DATA_BLOCK "dbMasterData"   // DB35
{ S7_Optimized_Access := 'FALSE' }
VERSION : 0.1
// stored: AutoNumber false, DBAccessibleFromOPCUA true, IsOnlyStoredInLoadMemory false, IsWriteProtectedInAS false
   VAR
      data5_Wielkość_przeływu_Adres_0 { S7_SetPoint := 'True'} : "typeDataMPP04_Int";   // wielkość przepływu / Wartość aktualnego przepływu
      data5_Licznik_objętość_VF_Adres_2 : "typeDataMPP04_Int";   // licznik objętości VF / Stan licznika objętości dla przepływu w przód VF
      data5_Licznik_objętość_VR_Adres_4 { S7_SetPoint := 'True'} : "typeDataMPP04_Int";   // licznik objętości VR / Stan licznika objętości dla przepływu w tył VR
      data5_Licznik_różnicowy_VD_Adres_6 { S7_SetPoint := 'True'} : "typeDataMPP04_Int";   // licznik różnicy / Stan bieżącego różnicowego licznika objętości VD
      data5_Stan_licz_bjętości_GF_Adres_8 { S7_SetPoint := 'True'} : "typeDataMPP04_Int";   // licznik objetosci GF / Stan głównego licznika objętości dla przepływu w przód GF
      data5_Stan_licz_bjętości_GR_Adres_10 { S7_SetPoint := 'True'} : "typeDataMPP04_Int";   // licznik objetości GR / Sta ngłownego licznika objętości dla przepływu w tył GR
      data5_Stan_licz_rózicowego_obj_GD_Adres_12 { S7_SetPoint := 'True'} : "typeDataMPP04_Int";   // licznik róznicowy / Stan głownego licznika różnicowego GD
      data5_Stan_urządzenia_1000 { S7_SetPoint := 'True'} : "typeDataInverter_Word";   // stan urządzenia / 8-przekrodzony zakres pracy przetwornika, 20-otwarty obwód cewki, 21zwarcie w obwodzie cewki, 26-brak cieczy w czujniku
      data6_Wielkość_przeływu_Adres_0 { S7_SetPoint := 'True'} : "typeDataMPP04_Int";   // wielkość przepływu / Wartość aktualnego przepływu
      data6_Licznik_objętość_VF_Adres_2 { S7_SetPoint := 'True'} : "typeDataMPP04_Int";   // licznik objętości VF / Stan licznika objętości dla przepływu w przód VF
      data6_Licznik_objętość_VR_Adres_4 { S7_SetPoint := 'True'} : "typeDataMPP04_Int";   // licznik objętości VR / Stan licznika objętości dla przepływu w tył VR
      data6_Licznik_różnicowy_VD_Adres_6 { S7_SetPoint := 'True'} : "typeDataMPP04_Int";   // licznik różnicy / Stan bieżącego różnicowego licznika objętości VD
      data6_Stan_licz_bjętości_GF_Adres_8 { S7_SetPoint := 'True'} : "typeDataMPP04_Int";   // licznik objetosci GF / Stan głównego licznika objętości dla przepływu w przód GF
      data6_Stan_licz_bjętości_GR_Adres_10 { S7_SetPoint := 'True'} : "typeDataMPP04_Int";   // licznik objetości GR / Sta ngłownego licznika objętości dla przepływu w tył GR
      data6_Stan_licz_rózicowego_obj_GD_Adres_12 { S7_SetPoint := 'True'} : "typeDataMPP04_Int";   // licznik róznicowy / Stan głownego licznika różnicowego GD
      data6_Stan_urządzenia_1000 { S7_SetPoint := 'True'} : "typeDataInverter_Word";   // stan urządzenia / 8-przekrodzony zakres pracy przetwornika, 20-otwarty obwód cewki, 21zwarcie w obwodzie cewki, 26-brak cieczy w czujniku
      data26_Inver_Control_word_416000_Fal { S7_SetPoint := 'True'} : "typeDataInverter_Word";   // Sowo komtrolneCTW falownika [Uint16, index 0]
      data26_Inver_setpoint_ref_416020_Fal { S7_SetPoint := 'True'} : "typeDataInverter_Word";   // Słowo wartość zadana Hz [Int16, index -1]
      data26_Inver_Status_word_416030_Fal { S7_SetPoint := 'True'} : "typeDataInverter_Word";   // Słowo statusu STW falownika [Uint16, index 0]
      data26_Inver_Frequency_416130_Fal { S7_SetPoint := 'True'} : "typeDataInverter_Word";   // Słowo częstotliwość na wyjściu [Uint16, index -1]
      data26_Inver_MotorCurrent_416140_Fal { S7_SetPoint := 'True'} : "typeDataInverter_Word";   // Słowo częstotliwość na wyjściu [Uint16, index -2]
      data26_Inver_DC_Voltage_416300_Fal { S7_SetPoint := 'True'} : "typeDataInverter_Word";   // Słowo napięcia DC na szynie [Uint16, index 0]
      data26_Inver_Temp_416340_Fal { S7_SetPoint := 'True'} : "typeDataInverter_Word";   // Słowo temperatura invertera [Uint8, index 0]
      data26_Inver_NomCurrent_416360_Fal { S7_SetPoint := 'True'} : "typeDataInverter_Word";   // Słowo nominalna wartośc prądu falonika[Uint16, index -2]
      data26_Inver_MaxCurrent_416370_Fal { S7_SetPoint := 'True'} : "typeDataInverter_Word";   // Słowo max prąd falownika [Uint16, index -2]
      data26_Inver_InDigit_416600_Fal { S7_SetPoint := 'True'} : "typeDataInverter_Word";   // Słowo mampa wejść 18,19,27,33 [Uint16, index -0]
      data26_Inver_HourWork_415010_Fal { S7_SetPoint := 'True'} : "typeDataInverter_DWord";   // Podwójne słowo czasu pracy falownika [Int32, index -0]
      data26_Inver_OverTemp_415040_Fal { S7_SetPoint := 'True'} : "typeDataInverter_Word";   // Sowo statusu przekroczenie temperatury[Uint16, index 0]
      data26_Inver_OverVolts_415050_Fal { S7_SetPoint := 'True'} : "typeDataInverter_Word";   // Sowo statusu przekroczenie napięcia[Uint16, index 0]
      data_RTU_value_0 { S7_SetPoint := 'True'} : "typeDataMPP04_real";   // Wartość 0.0 pomocnicza wyświetlana podczas błędu pomiaru
   END_VAR
BEGIN
   data_RTU_value_0.data[0] := 0.0;
END_DATA_BLOCK

DATA_BLOCK "dbModbusRTU_Reg"   // DB37
TITLE = Modbus RTU Data
{ S7_Optimized_Access := 'FALSE' }
AUTHOR : RTecmer
VERSION : 0.1
// Dane pomiarowe przekazane z bloku danych master modbus RTU
// stored: AutoNumber true, DBAccessibleFromOPCUA true, IsOnlyStoredInLoadMemory false, IsWriteProtectedInAS false
   VAR
      received_6_Wielkość_przeływu_Adres_0 { S7_SetPoint := 'True'} : "typeDataMPP04_Int";   // wielkość przepływu
      received_6_Licznik_objętość_VF_Adres_2 { S7_SetPoint := 'True'} : "typeDataMPP04_Int";   // licznik objętości VF
      received_6_Licznik_objętość_VR_Adres_4 { S7_SetPoint := 'True'} : "typeDataMPP04_Int";   // licznik objętości VR
      received_6_Licznik_różnicowy_VD_Adres_6 { S7_SetPoint := 'True'} : "typeDataMPP04_Int";   // licznik różnicy
      receive_6_Stan_licz_bjętości_GF_Adres_8 { S7_SetPoint := 'True'} : "typeDataMPP04_Int";   // licznik objetosci GF
      received_6_Stan_licz_bjętości_GR_Adres_10 { S7_SetPoint := 'True'} : "typeDataMPP04_Int";   // licznik objetości GR
      received_6_Stan_licz_rózicowego_obj_GD_Adres_12 { S7_SetPoint := 'True'} : "typeDataMPP04_Int";   // licznik róznicowy
      received_6_Stan_urządzenia_1000 { S7_SetPoint := 'True'} : "typeDataInverter_Word";   // stan urządzenia
      "Przepływomierz nr2" : Struct
         received_6_przeływu_VF_Adres_0 { S7_SetPoint := 'True'} : Real;
         received_6_objętość_VF_Adres_2 { S7_SetPoint := 'True'} : Real;
         "received_6_objętośc RF_Adres_4" { S7_SetPoint := 'True'} : Real;
         received_6_licznik_różnicowy_VD_Adres_7 { S7_SetPoint := 'True'} : Real;
         received_6_licznik_objętości_GF_Adres_8 { S7_SetPoint := 'True'} : Real;
         received_6_Licznik_objętości_GR_Adres_10 { S7_SetPoint := 'True'} : Real;
         received_6_Licznik_różnicowy_GD_Adres_12 { S7_SetPoint := 'True'} : Real;
         received_6_status_przepływomierza_Adres_1000 { S7_SetPoint := 'True'} : Word;
      END_STRUCT;
   END_VAR
BEGIN
END_DATA_BLOCK

DATA_BLOCK "dbTags_master_MPP04_2"   // DB81
{ S7_Optimized_Access := 'FALSE' }
VERSION : 0.1
// stored: AutoNumber true, DBAccessibleFromOPCUA true, IsOnlyStoredInLoadMemory false, IsWriteProtectedInAS false
   VAR
      "step" : USInt := 1;
      edge : Bool := false;
      modbusCommLoad { S7_SetPoint := 'True'} : "typeModbusCommLoad";
      modbusMaster { S7_SetPoint := 'True'} : "typeModbusMaster";
   END_VAR
BEGIN
END_DATA_BLOCK

DATA_BLOCK "dbTags_master_RTU"   // DB90
TITLE = Master
{ S7_Optimized_Access := 'FALSE' }
AUTHOR : rtecmer
VERSION : 0.1
// Instancja dla funkcji Mdbus RTU komunikacja z masterem MT101
// stored: AutoNumber false, DBAccessibleFromOPCUA true, IsOnlyStoredInLoadMemory false, IsWriteProtectedInAS false
   VAR
      "step" : USInt := 1;
      edge : Bool := false;
      modbusCommLoad { S7_SetPoint := 'True'} : "typeModbusCommLoad";
      modbusMaster { S7_SetPoint := 'True'} : "typeModbusSlave";
   END_VAR
BEGIN
   modbusMaster.mbAddr := 5;
END_DATA_BLOCK

ORGANIZATION_BLOCK "Main"   // OB1, LAD, ProgramCycle
TITLE = "Main Program Sweep (Cycle)"
{ S7_Optimized_Access := 'TRUE' }
VERSION : 0.1
// stored: AutoNumber true, IsIECCheckEnabled false, SetENOAutomatically false
   VAR_INPUT
      Initial_Call : Bool;   // Initial call of this OB
      Remanence : Bool;   // =True, if remanent data are available
   END_VAR
   VAR_TEMP   // added for the SCL form of the ladder/FBD networks
      _w1 : Bool;
      _w2 : Bool;
   END_VAR
BEGIN

REGION Network 1: Diagnostyka przerwań
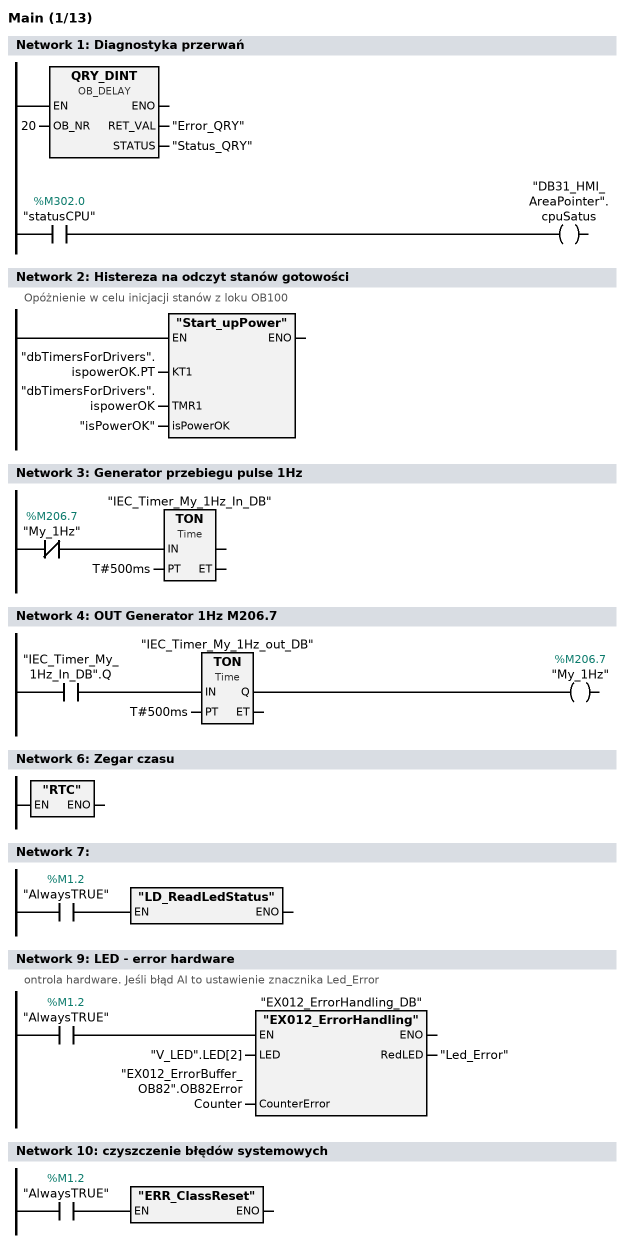
   RUNG wire#powerrail
      { S7_Templates := "obnr_type := OB_DELAY" } QRY_DINT(OB_NR := 20, RET_VAL => "Error_QRY", STATUS => "Status_QRY")
   END_RUNG
   RUNG wire#powerrail
      Contact( "statusCPU" )
      Coil( "DB31_HMI_AreaPointer".cpuSatus )
   END_RUNG
   // the same network as SCL:
   "Error_QRY" := QRY_DINT(OB_NR := 20, STATUS => "Status_QRY");
   "DB31_HMI_AreaPointer".cpuSatus := "statusCPU";
END_REGION

REGION Network 2: Histereza na odczyt stanów gotowości
   // Opóżnienie w celu inicjacji stanów z loku OB100
   RUNG wire#powerrail
      "Start_upPower"(KT1 := "dbTimersForDrivers".ispowerOK.PT, TMR1 := "dbTimersForDrivers".ispowerOK, isPowerOK := "isPowerOK")
   END_RUNG
   // the same network as SCL:
   "Start_upPower"(KT1 := "dbTimersForDrivers".ispowerOK.PT,
                   TMR1 := "dbTimersForDrivers".ispowerOK,
                   isPowerOK := "isPowerOK");
END_REGION

REGION Network 3: Generator przebiegu pulse 1Hz
   RUNG wire#powerrail
      I_Contact( "My_1Hz" )
      { S7_Templates := "time_type := Time" } "IEC_Timer_My_1Hz_In_DB".TON(pt := T#500ms, et =>)
   END_RUNG
   // the same network as SCL:
   "IEC_Timer_My_1Hz_In_DB".TON(IN := NOT "My_1Hz", PT := T#500ms);
END_REGION

REGION Network 4: OUT Generator 1Hz M206.7
   RUNG wire#powerrail
      Contact( "IEC_Timer_My_1Hz_In_DB".Q )
      { S7_Templates := "time_type := Time" } "IEC_Timer_My_1Hz_out_DB".TON(pt := T#500ms, et =>)
      Coil( "My_1Hz" )
   END_RUNG
   // the same network as SCL:
   "IEC_Timer_My_1Hz_out_DB".TON(IN := "IEC_Timer_My_1Hz_In_DB".Q, PT := T#500ms);
   "My_1Hz" := "IEC_Timer_My_1Hz_out_DB".Q;
END_REGION

REGION Network 6: Zegar czasu
   RUNG wire#powerrail
      "RTC"()
   END_RUNG
   // the same network as SCL:
   "RTC"();
END_REGION

REGION Network 7
   RUNG wire#powerrail
      Contact( "AlwaysTRUE" )
      "LD_ReadLedStatus"()
   END_RUNG
   // the same network as SCL:
   IF "AlwaysTRUE" THEN "LD_ReadLedStatus"(); END_IF;
END_REGION

REGION Network 8 (SCL): LED kontrola RUN
   // Przekazanie  stanu LED 1 CPU
   "DB31_HMI_AreaPointer".getPLCMode := "V_LED".LED[1];
END_REGION

REGION Network 9: LED - error hardware
   // ontrola hardware. Jeśli błąd AI to ustawienie znacznika Led_Error
   RUNG wire#powerrail
      Contact( "AlwaysTRUE" )
      "EX012_ErrorHandling_DB"(LED := "V_LED".LED[2], CounterError := "EX012_ErrorBuffer_OB82".OB82ErrorCounter, RedLED => "Led_Error")
   END_RUNG
   // the same network as SCL:
   IF "AlwaysTRUE" THEN
       "EX012_ErrorHandling_DB"(LED := "V_LED".LED[2],   // "EX012_ErrorHandling"
                               CounterError := "EX012_ErrorBuffer_OB82".OB82ErrorCounter,
                               RedLED => "Led_Error");
   END_IF;
END_REGION

REGION Network 10: czyszczenie błędów systemowych
   RUNG wire#powerrail
      Contact( "AlwaysTRUE" )
      "ERR_ClassReset"()
   END_RUNG
   // the same network as SCL:
   IF "AlwaysTRUE" THEN "ERR_ClassReset"(); END_IF;
END_REGION

REGION Network 11: kontrola błedów
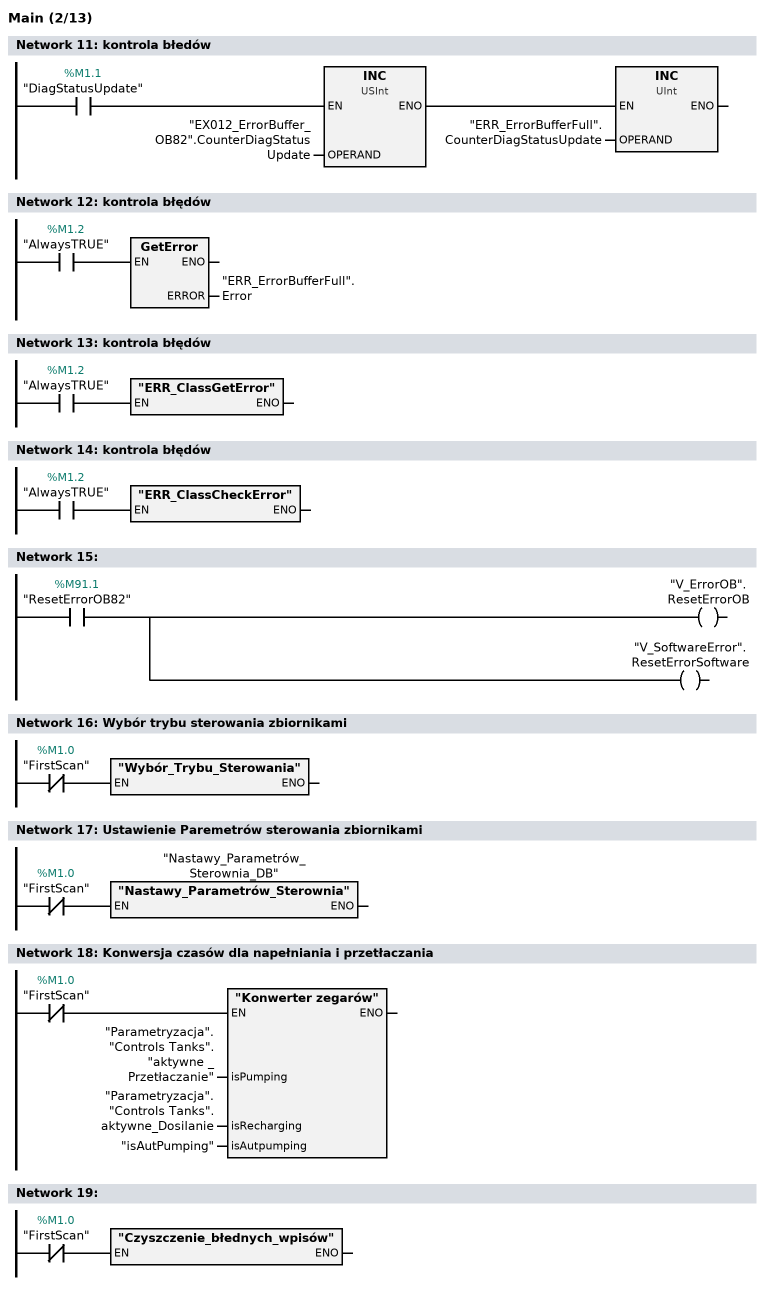
   RUNG wire#powerrail
      Contact( "DiagStatusUpdate" )
      { S7_Templates := "DestType := USInt" } Inc( "EX012_ErrorBuffer_OB82".CounterDiagStatusUpdate )
      { S7_Templates := "DestType := UInt" } Inc( "ERR_ErrorBufferFull".CounterDiagStatusUpdate )
   END_RUNG
   // the same network as SCL:
   IF "DiagStatusUpdate" THEN
       "EX012_ErrorBuffer_OB82".CounterDiagStatusUpdate := "EX012_ErrorBuffer_OB82".CounterDiagStatusUpdate + 1;
       "ERR_ErrorBufferFull".CounterDiagStatusUpdate := "ERR_ErrorBufferFull".CounterDiagStatusUpdate + 1;
   END_IF;
END_REGION

REGION Network 12: kontrola błędów
   // no SCL statement known for GetError: written as a call
   IF "AlwaysTRUE" THEN GetError(error => "ERR_ErrorBufferFull".Error); END_IF;
END_REGION

REGION Network 13: kontrola błędów
   RUNG wire#powerrail
      Contact( "AlwaysTRUE" )
      "ERR_ClassGetError"()
   END_RUNG
   // the same network as SCL:
   IF "AlwaysTRUE" THEN "ERR_ClassGetError"(); END_IF;
END_REGION

REGION Network 14: kontrola błędów
   RUNG wire#powerrail
      Contact( "AlwaysTRUE" )
      "ERR_ClassCheckError"()
   END_RUNG
   // the same network as SCL:
   IF "AlwaysTRUE" THEN "ERR_ClassCheckError"(); END_IF;
END_REGION

REGION Network 15
   RUNG wire#powerrail
      Contact( "ResetErrorOB82" )
      wire#w1
      Coil( "V_ErrorOB".ResetErrorOB )
   END_RUNG
   RUNG wire#w1
      Coil( "V_SoftwareError".ResetErrorSoftware )
   END_RUNG
   // the same network as SCL:
   "V_ErrorOB".ResetErrorOB := "ResetErrorOB82";
   "V_SoftwareError".ResetErrorSoftware := "ResetErrorOB82";
END_REGION

REGION Network 16: Wybór trybu sterowania zbiornikami
   RUNG wire#powerrail
      I_Contact( "FirstScan" )
      "Wybór_Trybu_Sterowania"()
   END_RUNG
   // the same network as SCL:
   IF NOT "FirstScan" THEN "Wybór_Trybu_Sterowania"(); END_IF;
END_REGION

REGION Network 17: Ustawienie Paremetrów sterowania zbiornikami
   RUNG wire#powerrail
      I_Contact( "FirstScan" )
      "Nastawy_Parametrów_Sterownia_DB"()
   END_RUNG
   // the same network as SCL:
   IF NOT "FirstScan" THEN
       "Nastawy_Parametrów_Sterownia_DB"();   // "Nastawy_Parametrów_Sterownia"
   END_IF;
END_REGION

REGION Network 18: Konwersja czasów dla napełniania i przetłaczania
   RUNG wire#powerrail
      I_Contact( "FirstScan" )
      "Konwerter zegarów"(isPumping := "Parametryzacja"."Controls Tanks"."aktywne _Przetłaczanie", isRecharging := "Parametryzacja"."Controls Tanks".aktywne_Dosilanie, isAutpumping := "isAutPumping")
   END_RUNG
   // the same network as SCL:
   IF NOT "FirstScan" THEN
       "Konwerter zegarów"(isPumping := "Parametryzacja"."Controls Tanks"."aktywne _Przetłaczanie",
                           isRecharging := "Parametryzacja"."Controls Tanks".aktywne_Dosilanie,
                           isAutpumping := "isAutPumping");
   END_IF;
END_REGION

REGION Network 19
   RUNG wire#powerrail
      I_Contact( "FirstScan" )
      "Czyszczenie_błednych_wpisów"()
   END_RUNG
   // the same network as SCL:
   IF NOT "FirstScan" THEN "Czyszczenie_błednych_wpisów"(); END_IF;
END_REGION

REGION Network 20: Modbus RTU
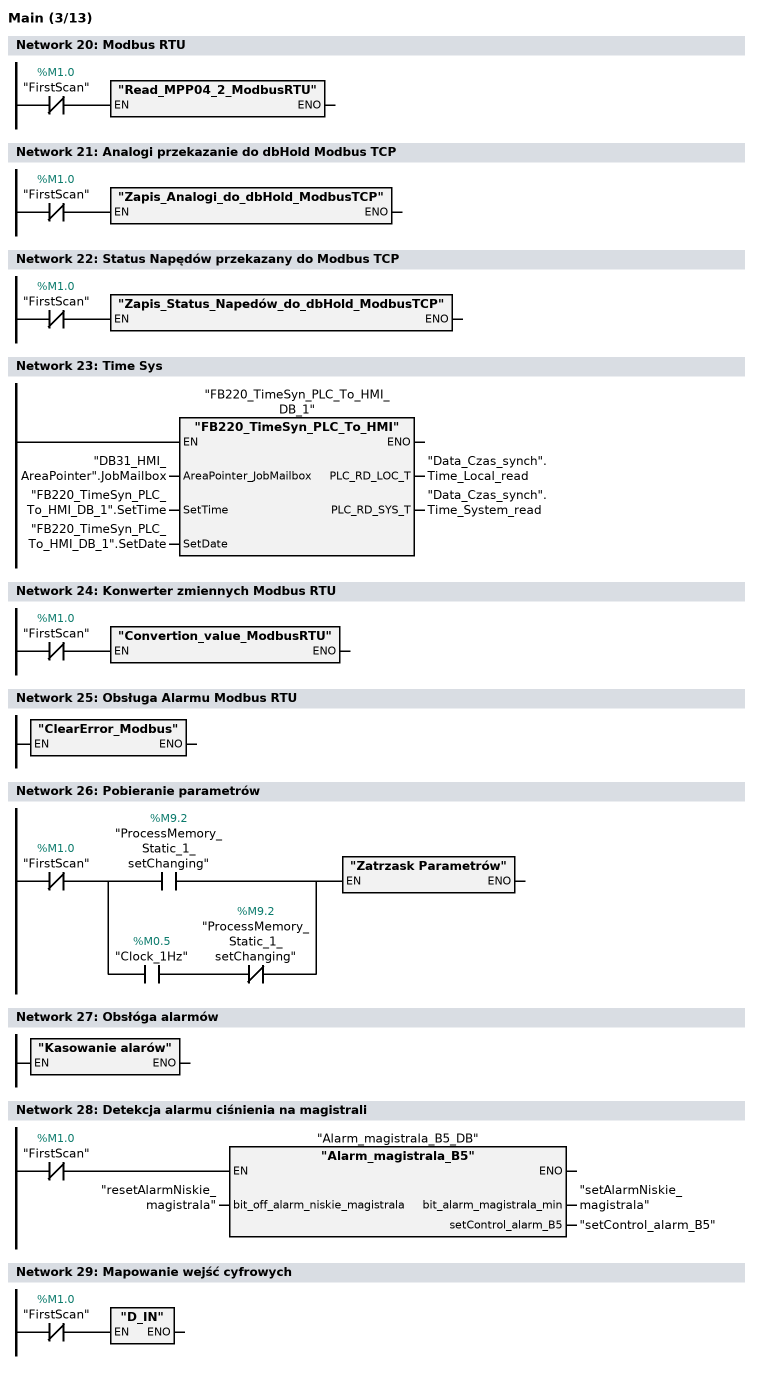
   RUNG wire#powerrail
      I_Contact( "FirstScan" )
      "Read_MPP04_2_ModbusRTU"()
   END_RUNG
   // the same network as SCL:
   IF NOT "FirstScan" THEN "Read_MPP04_2_ModbusRTU"(); END_IF;
END_REGION

REGION Network 21: Analogi przekazanie do dbHold Modbus TCP
   RUNG wire#powerrail
      I_Contact( "FirstScan" )
      "Zapis_Analogi_do_dbHold_ModbusTCP"()
   END_RUNG
   // the same network as SCL:
   IF NOT "FirstScan" THEN "Zapis_Analogi_do_dbHold_ModbusTCP"(); END_IF;
END_REGION

REGION Network 22: Status Napędów przekazany do Modbus TCP
   RUNG wire#powerrail
      I_Contact( "FirstScan" )
      "Zapis_Status_Napedów_do_dbHold_ModbusTCP"()
   END_RUNG
   // the same network as SCL:
   IF NOT "FirstScan" THEN "Zapis_Status_Napedów_do_dbHold_ModbusTCP"(); END_IF;
END_REGION

REGION Network 23: Time Sys
   RUNG wire#powerrail
      "FB220_TimeSyn_PLC_To_HMI_DB_1"(AreaPointer_JobMailbox := "DB31_HMI_AreaPointer".JobMailbox, SetTime := "FB220_TimeSyn_PLC_To_HMI_DB_1".SetTime, SetDate := "FB220_TimeSyn_PLC_To_HMI_DB_1".SetDate, PLC_RD_LOC_T => "Data_Czas_synch".Time_Local_read, PLC_RD_SYS_T => "Data_Czas_synch".Time_System_read)
   END_RUNG
   // the same network as SCL:
   "FB220_TimeSyn_PLC_To_HMI_DB_1"(AreaPointer_JobMailbox := "DB31_HMI_AreaPointer".JobMailbox,   // "FB220_TimeSyn_PLC_To_HMI"
                           SetTime := "FB220_TimeSyn_PLC_To_HMI_DB_1".SetTime,
                           SetDate := "FB220_TimeSyn_PLC_To_HMI_DB_1".SetDate,
                           PLC_RD_LOC_T => "Data_Czas_synch".Time_Local_read,
                           PLC_RD_SYS_T => "Data_Czas_synch".Time_System_read);
END_REGION

REGION Network 24: Konwerter zmiennych Modbus RTU
   RUNG wire#powerrail
      I_Contact( "FirstScan" )
      "Convertion_value_ModbusRTU"()
   END_RUNG
   // the same network as SCL:
   IF NOT "FirstScan" THEN "Convertion_value_ModbusRTU"(); END_IF;
END_REGION

REGION Network 25: Obsługa Alarmu Modbus RTU
   RUNG wire#powerrail
      "ClearError_Modbus"()
   END_RUNG
   // the same network as SCL:
   "ClearError_Modbus"();
END_REGION

REGION Network 26: Pobieranie parametrów
   RUNG wire#powerrail
      I_Contact( "FirstScan" )
      wire#w1
      Contact( "ProcessMemory_Static_1_setChanging" )
      wire#w2
      "Zatrzask Parametrów"()
   END_RUNG
   RUNG wire#w1
      Contact( "Clock_1Hz" )
      I_Contact( "ProcessMemory_Static_1_setChanging" )
   END_RUNG wire#w2
   // the same network as SCL:
   IF NOT "FirstScan" AND ("ProcessMemory_Static_1_setChanging" OR ("Clock_1Hz" AND NOT "ProcessMemory_Static_1_setChanging")) THEN
       "Zatrzask Parametrów"();
   END_IF;
END_REGION

REGION Network 27: Obsłóga alarmów
   RUNG wire#powerrail
      "Kasowanie alarów"()
   END_RUNG
   // the same network as SCL:
   "Kasowanie alarów"();
END_REGION

REGION Network 28: Detekcja alarmu ciśnienia na magistrali
   RUNG wire#powerrail
      I_Contact( "FirstScan" )
      "Alarm_magistrala_B5_DB"(bit_off_alarm_niskie_magistrala := "resetAlarmNiskie_magistrala", bit_alarm_magistrala_min => "setAlarmNiskie_magistrala", setControl_alarm_B5 => "setControl_alarm_B5")
   END_RUNG
   // the same network as SCL:
   IF NOT "FirstScan" THEN
       "Alarm_magistrala_B5_DB"(bit_off_alarm_niskie_magistrala := "resetAlarmNiskie_magistrala",   // "Alarm_magistrala_B5"
                               bit_alarm_magistrala_min => "setAlarmNiskie_magistrala",
                               setControl_alarm_B5 => "setControl_alarm_B5");
   END_IF;
END_REGION

REGION Network 29: Mapowanie wejść cyfrowych
   RUNG wire#powerrail
      I_Contact( "FirstScan" )
      "D_IN"()
   END_RUNG
   // the same network as SCL:
   IF NOT "FirstScan" THEN "D_IN"(); END_IF;
END_REGION

REGION Network 30: Wejścia Analogowe
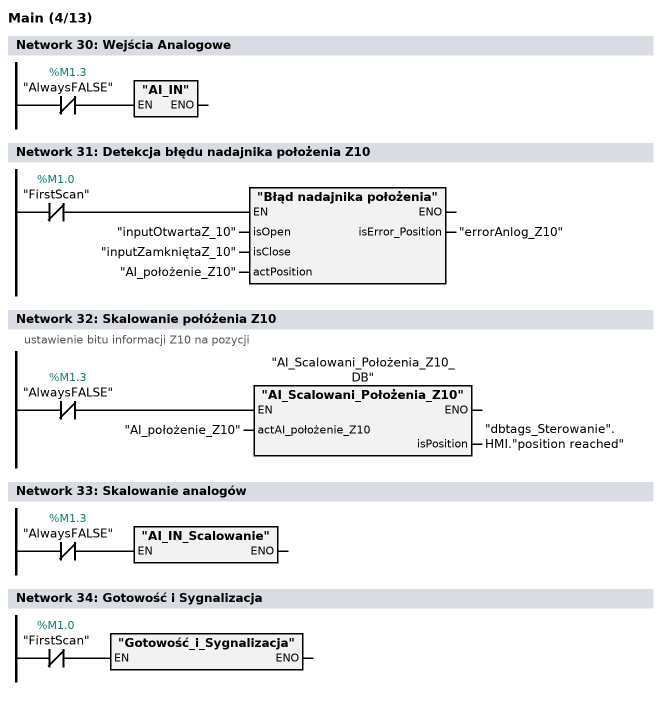
   RUNG wire#powerrail
      I_Contact( "AlwaysFALSE" )
      "AI_IN"()
   END_RUNG
   // the same network as SCL:
   IF NOT "AlwaysFALSE" THEN "AI_IN"(); END_IF;
END_REGION

REGION Network 31: Detekcja błędu nadajnika położenia Z10
   RUNG wire#powerrail
      I_Contact( "FirstScan" )
      "Błąd nadajnika położenia"(isOpen := "inputOtwartaZ_10", isClose := "inputZamkniętaZ_10", actPosition := "AI_położenie_Z10", isError_Position => "errorAnlog_Z10")
   END_RUNG
   // the same network as SCL:
   IF NOT "FirstScan" THEN
       "Błąd nadajnika położenia"(isOpen := "inputOtwartaZ_10",
                               isClose := "inputZamkniętaZ_10",
                               actPosition := "AI_położenie_Z10",
                               isError_Position => "errorAnlog_Z10");
   END_IF;
END_REGION

REGION Network 32: Skalowanie połóżenia Z10
   // ustawienie bitu informacji Z10 na pozycji
   RUNG wire#powerrail
      I_Contact( "AlwaysFALSE" )
      "AI_Scalowani_Położenia_Z10_DB"(actAI_położenie_Z10 := "AI_położenie_Z10", isPosition => "dbtags_Sterowanie".HMI."position reached")
   END_RUNG
   // the same network as SCL:
   IF NOT "AlwaysFALSE" THEN
       "AI_Scalowani_Położenia_Z10_DB"(actAI_położenie_Z10 := "AI_położenie_Z10",   // "AI_Scalowani_Położenia_Z10"
                               isPosition => "dbtags_Sterowanie".HMI."position reached");
   END_IF;
END_REGION

REGION Network 33: Skalowanie analogów
   RUNG wire#powerrail
      I_Contact( "AlwaysFALSE" )
      "AI_IN_Scalowanie"()
   END_RUNG
   // the same network as SCL:
   IF NOT "AlwaysFALSE" THEN "AI_IN_Scalowanie"(); END_IF;
END_REGION

REGION Network 34: Gotowość i Sygnalizacja
   RUNG wire#powerrail
      I_Contact( "FirstScan" )
      "Gotowość_i_Sygnalizacja"()
   END_RUNG
   // the same network as SCL:
   IF NOT "FirstScan" THEN "Gotowość_i_Sygnalizacja"(); END_IF;
END_REGION

REGION Network 35
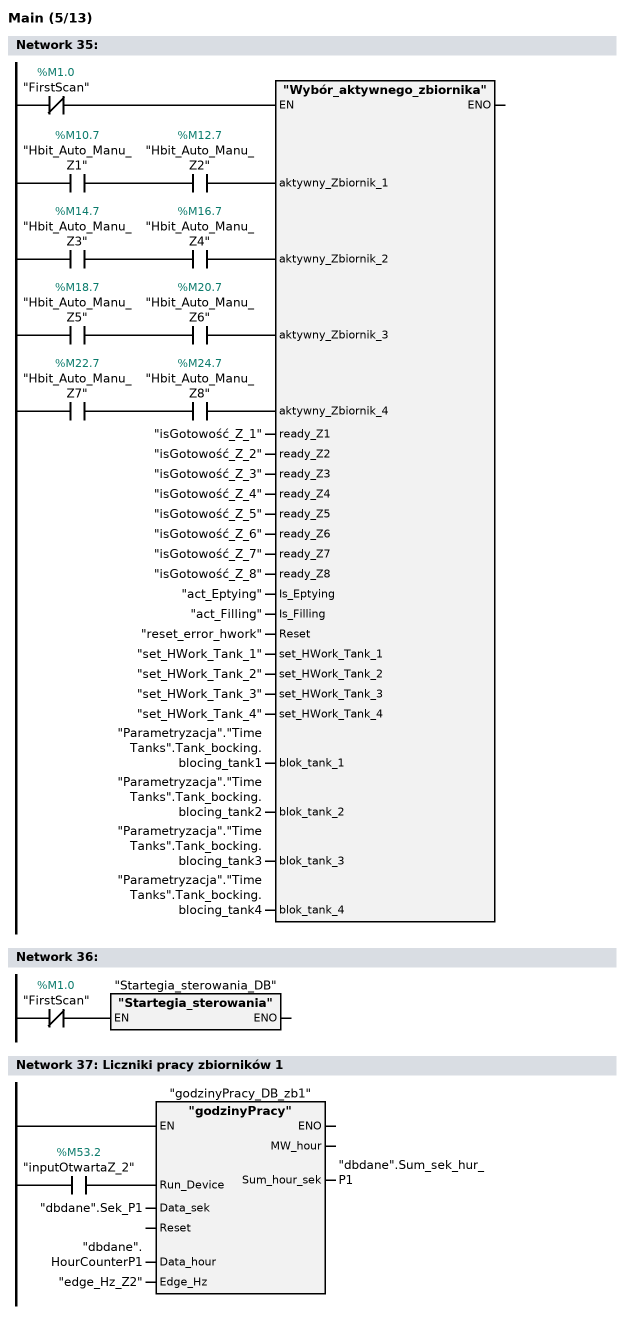
   RUNG wire#powerrail
      I_Contact( "FirstScan" )
      "Wybór_aktywnego_zbiornika"(aktywny_Zbiornik_1 := wire#w1, aktywny_Zbiornik_2 := wire#w2, aktywny_Zbiornik_3 := wire#w3, aktywny_Zbiornik_4 := wire#w4, ready_Z1 := "isGotowość_Z_1", ready_Z2 := "isGotowość_Z_2", ready_Z3 := "isGotowość_Z_3", ready_Z4 := "isGotowość_Z_4", ready_Z5 := "isGotowość_Z_5", ready_Z6 := "isGotowość_Z_6", ready_Z7 := "isGotowość_Z_7", ready_Z8 := "isGotowość_Z_8", Is_Eptying := "act_Eptying", Is_Filling := "act_Filling", Reset := "reset_error_hwork", set_HWork_Tank_1 := "set_HWork_Tank_1", set_HWork_Tank_2 := "set_HWork_Tank_2", set_HWork_Tank_3 := "set_HWork_Tank_3", set_HWork_Tank_4 := "set_HWork_Tank_4", blok_tank_1 := "Parametryzacja"."Time Tanks".Tank_bocking.blocing_tank1, blok_tank_2 := "Parametryzacja"."Time Tanks".Tank_bocking.blocing_tank2, blok_tank_3 := "Parametryzacja"."Time Tanks".Tank_bocking.blocing_tank3, blok_tank_4 := "Parametryzacja"."Time Tanks".Tank_bocking.blocing_tank4)
   END_RUNG
   RUNG wire#powerrail
      Contact( "Hbit_Auto_Manu_Z1" )
      Contact( "Hbit_Auto_Manu_Z2" )
   END_RUNG wire#w1
   RUNG wire#powerrail
      Contact( "Hbit_Auto_Manu_Z3" )
      Contact( "Hbit_Auto_Manu_Z4" )
   END_RUNG wire#w2
   RUNG wire#powerrail
      Contact( "Hbit_Auto_Manu_Z5" )
      Contact( "Hbit_Auto_Manu_Z6" )
   END_RUNG wire#w3
   RUNG wire#powerrail
      Contact( "Hbit_Auto_Manu_Z7" )
      Contact( "Hbit_Auto_Manu_Z8" )
   END_RUNG wire#w4
   // the same network as SCL:
   IF NOT "FirstScan" THEN
       "Wybór_aktywnego_zbiornika"(aktywny_Zbiornik_1 := "Hbit_Auto_Manu_Z1" AND "Hbit_Auto_Manu_Z2",
                               aktywny_Zbiornik_2 := "Hbit_Auto_Manu_Z3" AND "Hbit_Auto_Manu_Z4",
                               aktywny_Zbiornik_3 := "Hbit_Auto_Manu_Z5" AND "Hbit_Auto_Manu_Z6",
                               aktywny_Zbiornik_4 := "Hbit_Auto_Manu_Z7" AND "Hbit_Auto_Manu_Z8",
                               ready_Z1 := "isGotowość_Z_1",
                               ready_Z2 := "isGotowość_Z_2",
                               ready_Z3 := "isGotowość_Z_3",
                               ready_Z4 := "isGotowość_Z_4",
                               ready_Z5 := "isGotowość_Z_5",
                               ready_Z6 := "isGotowość_Z_6",
                               ready_Z7 := "isGotowość_Z_7",
                               ready_Z8 := "isGotowość_Z_8",
                               Is_Eptying := "act_Eptying",
                               Is_Filling := "act_Filling",
                               Reset := "reset_error_hwork",
                               set_HWork_Tank_1 := "set_HWork_Tank_1",
                               set_HWork_Tank_2 := "set_HWork_Tank_2",
                               set_HWork_Tank_3 := "set_HWork_Tank_3",
                               set_HWork_Tank_4 := "set_HWork_Tank_4",
                               blok_tank_1 := "Parametryzacja"."Time Tanks".Tank_bocking.blocing_tank1,
                               blok_tank_2 := "Parametryzacja"."Time Tanks".Tank_bocking.blocing_tank2,
                               blok_tank_3 := "Parametryzacja"."Time Tanks".Tank_bocking.blocing_tank3,
                               blok_tank_4 := "Parametryzacja"."Time Tanks".Tank_bocking.blocing_tank4);
   END_IF;
END_REGION

REGION Network 36
   RUNG wire#powerrail
      I_Contact( "FirstScan" )
      "Startegia_sterowania_DB"()
   END_RUNG
   // the same network as SCL:
   IF NOT "FirstScan" THEN
       "Startegia_sterowania_DB"();   // "Startegia_sterowania"
   END_IF;
END_REGION

REGION Network 37: Liczniki pracy zbiorników 1
   RUNG wire#powerrail
      "godzinyPracy_DB_zb1"(Run_Device := wire#w1, Data_sek := "dbdane".Sek_P1, Reset :=, Data_hour := "dbdane".HourCounterP1, Edge_Hz := "edge_Hz_Z2", MW_hour =>, Sum_hour_sek => "dbdane".Sum_sek_hur_P1)
   END_RUNG
   RUNG wire#powerrail
      Contact( "inputOtwartaZ_2" )
   END_RUNG wire#w1
   // the same network as SCL:
   "godzinyPracy_DB_zb1"(Run_Device := "inputOtwartaZ_2",   // "godzinyPracy"
                         Data_sek := "dbdane".Sek_P1,
                         Data_hour := "dbdane".HourCounterP1,
                         Edge_Hz := "edge_Hz_Z2",
                         Sum_hour_sek => "dbdane".Sum_sek_hur_P1);
END_REGION

REGION Network 38: Liczniki pracy zbiorników 2
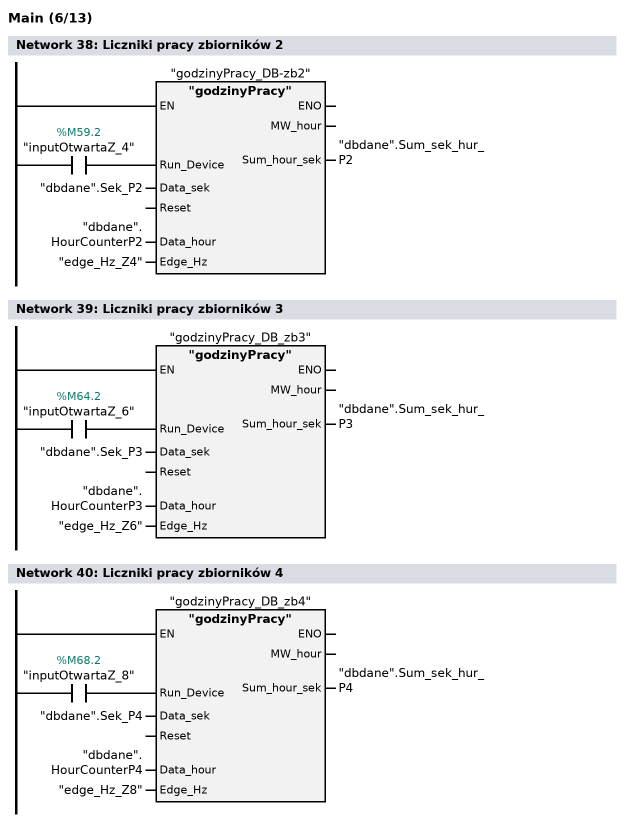
   RUNG wire#powerrail
      "godzinyPracy_DB-zb2"(Run_Device := wire#w1, Data_sek := "dbdane".Sek_P2, Reset :=, Data_hour := "dbdane".HourCounterP2, Edge_Hz := "edge_Hz_Z4", MW_hour =>, Sum_hour_sek => "dbdane".Sum_sek_hur_P2)
   END_RUNG
   RUNG wire#powerrail
      Contact( "inputOtwartaZ_4" )
   END_RUNG wire#w1
   // the same network as SCL:
   "godzinyPracy_DB-zb2"(Run_Device := "inputOtwartaZ_4",   // "godzinyPracy"
                         Data_sek := "dbdane".Sek_P2,
                         Data_hour := "dbdane".HourCounterP2,
                         Edge_Hz := "edge_Hz_Z4",
                         Sum_hour_sek => "dbdane".Sum_sek_hur_P2);
END_REGION

REGION Network 39: Liczniki pracy zbiorników 3
   RUNG wire#powerrail
      "godzinyPracy_DB_zb3"(Run_Device := wire#w1, Data_sek := "dbdane".Sek_P3, Reset :=, Data_hour := "dbdane".HourCounterP3, Edge_Hz := "edge_Hz_Z6", MW_hour =>, Sum_hour_sek => "dbdane".Sum_sek_hur_P3)
   END_RUNG
   RUNG wire#powerrail
      Contact( "inputOtwartaZ_6" )
   END_RUNG wire#w1
   // the same network as SCL:
   "godzinyPracy_DB_zb3"(Run_Device := "inputOtwartaZ_6",   // "godzinyPracy"
                         Data_sek := "dbdane".Sek_P3,
                         Data_hour := "dbdane".HourCounterP3,
                         Edge_Hz := "edge_Hz_Z6",
                         Sum_hour_sek => "dbdane".Sum_sek_hur_P3);
END_REGION

REGION Network 40: Liczniki pracy zbiorników 4
   RUNG wire#powerrail
      "godzinyPracy_DB_zb4"(Run_Device := wire#w1, Data_sek := "dbdane".Sek_P4, Reset :=, Data_hour := "dbdane".HourCounterP4, Edge_Hz := "edge_Hz_Z8", MW_hour =>, Sum_hour_sek => "dbdane".Sum_sek_hur_P4)
   END_RUNG
   RUNG wire#powerrail
      Contact( "inputOtwartaZ_8" )
   END_RUNG wire#w1
   // the same network as SCL:
   "godzinyPracy_DB_zb4"(Run_Device := "inputOtwartaZ_8",   // "godzinyPracy"
                         Data_sek := "dbdane".Sek_P4,
                         Data_hour := "dbdane".HourCounterP4,
                         Edge_Hz := "edge_Hz_Z8",
                         Sum_hour_sek => "dbdane".Sum_sek_hur_P4);
END_REGION

REGION Network 41: Sterowanie zbiornikami nr 1
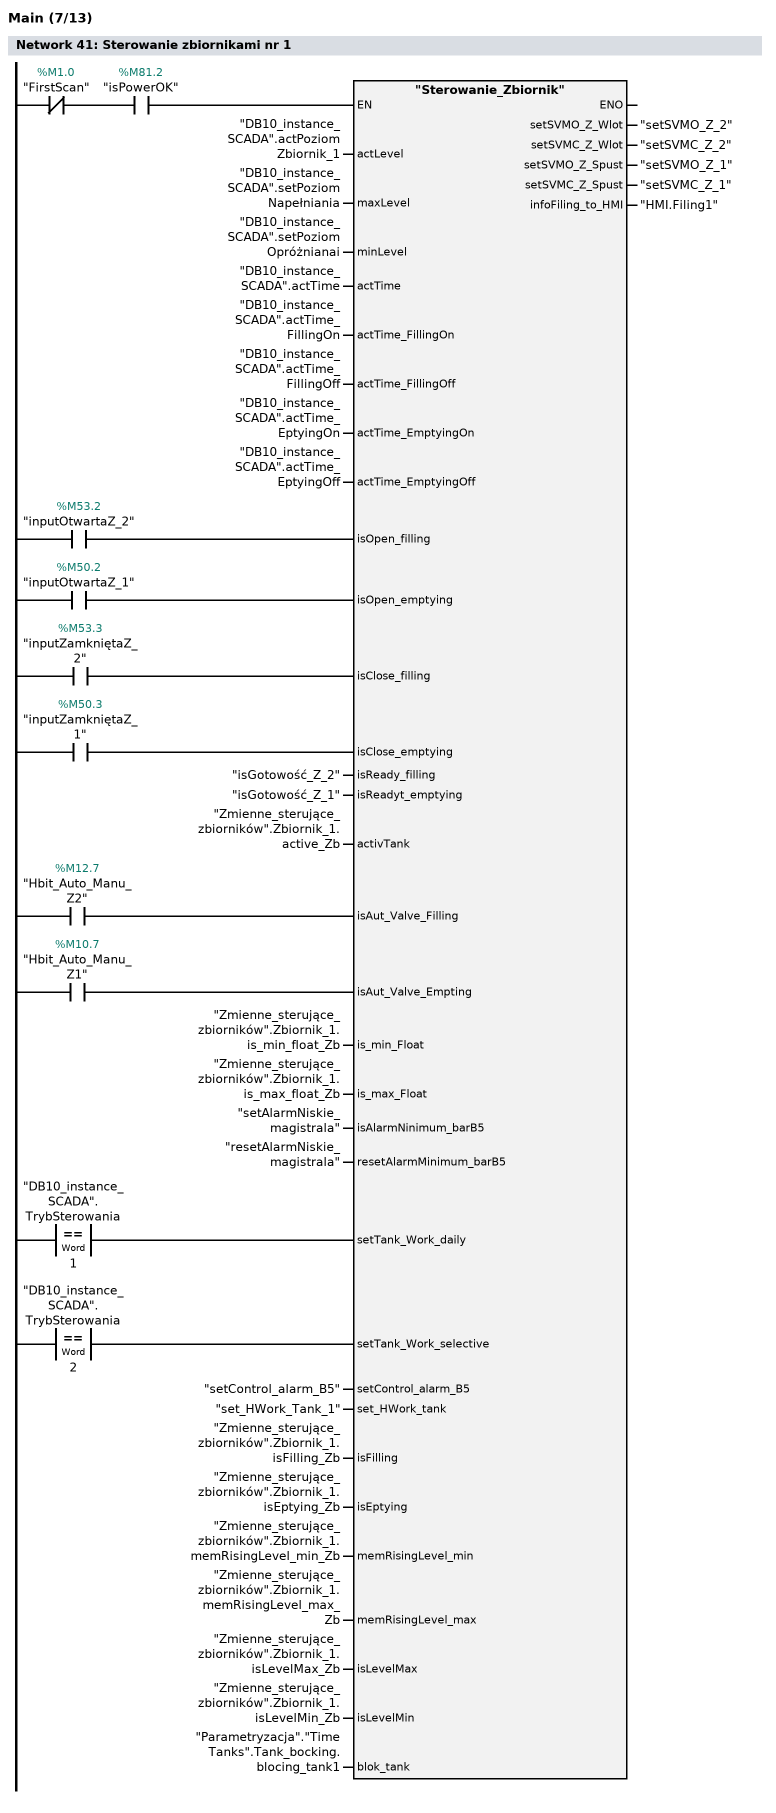
   RUNG wire#powerrail
      I_Contact( "FirstScan" )
      Contact( "isPowerOK" )
      "Sterowanie_Zbiornik"(isOpen_filling := wire#w1, isOpen_emptying := wire#w2, isClose_filling := wire#w3, isClose_emptying := wire#w4, isAut_Valve_Filling := wire#w5, isAut_Valve_Empting := wire#w6, setTank_Work_daily := wire#w7, setTank_Work_selective := wire#w8, actLevel := "DB10_instance_SCADA".actPoziomZbiornik_1, maxLevel := "DB10_instance_SCADA".setPoziomNapełniania, minLevel := "DB10_instance_SCADA".setPoziomOpróżnianai, actTime := "DB10_instance_SCADA".actTime, actTime_FillingOn := "DB10_instance_SCADA".actTime_FillingOn, actTime_FillingOff := "DB10_instance_SCADA".actTime_FillingOff, actTime_EmptyingOn := "DB10_instance_SCADA".actTime_EptyingOn, actTime_EmptyingOff := "DB10_instance_SCADA".actTime_EptyingOff, isReady_filling := "isGotowość_Z_2", isReadyt_emptying := "isGotowość_Z_1", activTank := "Zmienne_sterujące_zbiorników".Zbiornik_1.active_Zb, is_min_Float := "Zmienne_sterujące_zbiorników".Zbiornik_1.is_min_float_Zb, is_max_Float := "Zmienne_sterujące_zbiorników".Zbiornik_1.is_max_float_Zb, isAlarmNinimum_barB5 := "setAlarmNiskie_magistrala", resetAlarmMinimum_barB5 := "resetAlarmNiskie_magistrala", setControl_alarm_B5 := "setControl_alarm_B5", set_HWork_tank := "set_HWork_Tank_1", isFilling := "Zmienne_sterujące_zbiorników".Zbiornik_1.isFilling_Zb, isEptying := "Zmienne_sterujące_zbiorników".Zbiornik_1.isEptying_Zb, memRisingLevel_min := "Zmienne_sterujące_zbiorników".Zbiornik_1.memRisingLevel_min_Zb, memRisingLevel_max := "Zmienne_sterujące_zbiorników".Zbiornik_1.memRisingLevel_max_Zb, isLevelMax := "Zmienne_sterujące_zbiorników".Zbiornik_1.isLevelMax_Zb, isLevelMin := "Zmienne_sterujące_zbiorników".Zbiornik_1.isLevelMin_Zb, blok_tank := "Parametryzacja"."Time Tanks".Tank_bocking.blocing_tank1, setSVMO_Z_Wlot => "setSVMO_Z_2", setSVMC_Z_Wlot => "setSVMC_Z_2", setSVMO_Z_Spust => "setSVMO_Z_1", setSVMC_Z_Spust => "setSVMC_Z_1", infoFiling_to_HMI => "HMI.Filing1")
   END_RUNG
   RUNG wire#powerrail
      Contact( "inputOtwartaZ_2" )
   END_RUNG wire#w1
   RUNG wire#powerrail
      Contact( "inputOtwartaZ_1" )
   END_RUNG wire#w2
   RUNG wire#powerrail
      Contact( "inputZamkniętaZ_2" )
   END_RUNG wire#w3
   RUNG wire#powerrail
      Contact( "inputZamkniętaZ_1" )
   END_RUNG wire#w4
   RUNG wire#powerrail
      Contact( "Hbit_Auto_Manu_Z2" )
   END_RUNG wire#w5
   RUNG wire#powerrail
      Contact( "Hbit_Auto_Manu_Z1" )
   END_RUNG wire#w6
   RUNG wire#powerrail
      { S7_Templates := "SrcType := Word" } EQ_Contact(in1 := "DB10_instance_SCADA".TrybSterowania, in2 := 1)
   END_RUNG wire#w7
   RUNG wire#powerrail
      { S7_Templates := "SrcType := Word" } EQ_Contact(in1 := "DB10_instance_SCADA".TrybSterowania, in2 := 2)
   END_RUNG wire#w8
   // the same network as SCL:
   IF NOT "FirstScan" AND "isPowerOK" THEN
       "Sterowanie_Zbiornik"(actLevel := "DB10_instance_SCADA".actPoziomZbiornik_1,
                             maxLevel := "DB10_instance_SCADA".setPoziomNapełniania,
                             minLevel := "DB10_instance_SCADA".setPoziomOpróżnianai,
                             actTime := "DB10_instance_SCADA".actTime,
                             actTime_FillingOn := "DB10_instance_SCADA".actTime_FillingOn,
                             actTime_FillingOff := "DB10_instance_SCADA".actTime_FillingOff,
                             actTime_EmptyingOn := "DB10_instance_SCADA".actTime_EptyingOn,
                             actTime_EmptyingOff := "DB10_instance_SCADA".actTime_EptyingOff,
                             isOpen_filling := "inputOtwartaZ_2",
                             isOpen_emptying := "inputOtwartaZ_1",
                             isClose_filling := "inputZamkniętaZ_2",
                             isClose_emptying := "inputZamkniętaZ_1",
                             isReady_filling := "isGotowość_Z_2",
                             isReadyt_emptying := "isGotowość_Z_1",
                             activTank := "Zmienne_sterujące_zbiorników".Zbiornik_1.active_Zb,
                             isAut_Valve_Filling := "Hbit_Auto_Manu_Z2",
                             isAut_Valve_Empting := "Hbit_Auto_Manu_Z1",
                             is_min_Float := "Zmienne_sterujące_zbiorników".Zbiornik_1.is_min_float_Zb,
                             is_max_Float := "Zmienne_sterujące_zbiorników".Zbiornik_1.is_max_float_Zb,
                             isAlarmNinimum_barB5 := "setAlarmNiskie_magistrala",
                             resetAlarmMinimum_barB5 := "resetAlarmNiskie_magistrala",
                             setTank_Work_daily := "DB10_instance_SCADA".TrybSterowania = 1,
                             setTank_Work_selective := "DB10_instance_SCADA".TrybSterowania = 2,
                             setControl_alarm_B5 := "setControl_alarm_B5",
                             set_HWork_tank := "set_HWork_Tank_1",
                             isFilling := "Zmienne_sterujące_zbiorników".Zbiornik_1.isFilling_Zb,
                             isEptying := "Zmienne_sterujące_zbiorników".Zbiornik_1.isEptying_Zb,
                             memRisingLevel_min := "Zmienne_sterujące_zbiorników".Zbiornik_1.memRisingLevel_min_Zb,
                             memRisingLevel_max := "Zmienne_sterujące_zbiorników".Zbiornik_1.memRisingLevel_max_Zb,
                             isLevelMax := "Zmienne_sterujące_zbiorników".Zbiornik_1.isLevelMax_Zb,
                             isLevelMin := "Zmienne_sterujące_zbiorników".Zbiornik_1.isLevelMin_Zb,
                             blok_tank := "Parametryzacja"."Time Tanks".Tank_bocking.blocing_tank1,
                             setSVMO_Z_Wlot => "setSVMO_Z_2",
                             setSVMC_Z_Wlot => "setSVMC_Z_2",
                             setSVMO_Z_Spust => "setSVMO_Z_1",
                             setSVMC_Z_Spust => "setSVMC_Z_1",
                             infoFiling_to_HMI => "HMI.Filing1");
   END_IF;
END_REGION

REGION Network 42: Sterowanie zbiornikami nr 2
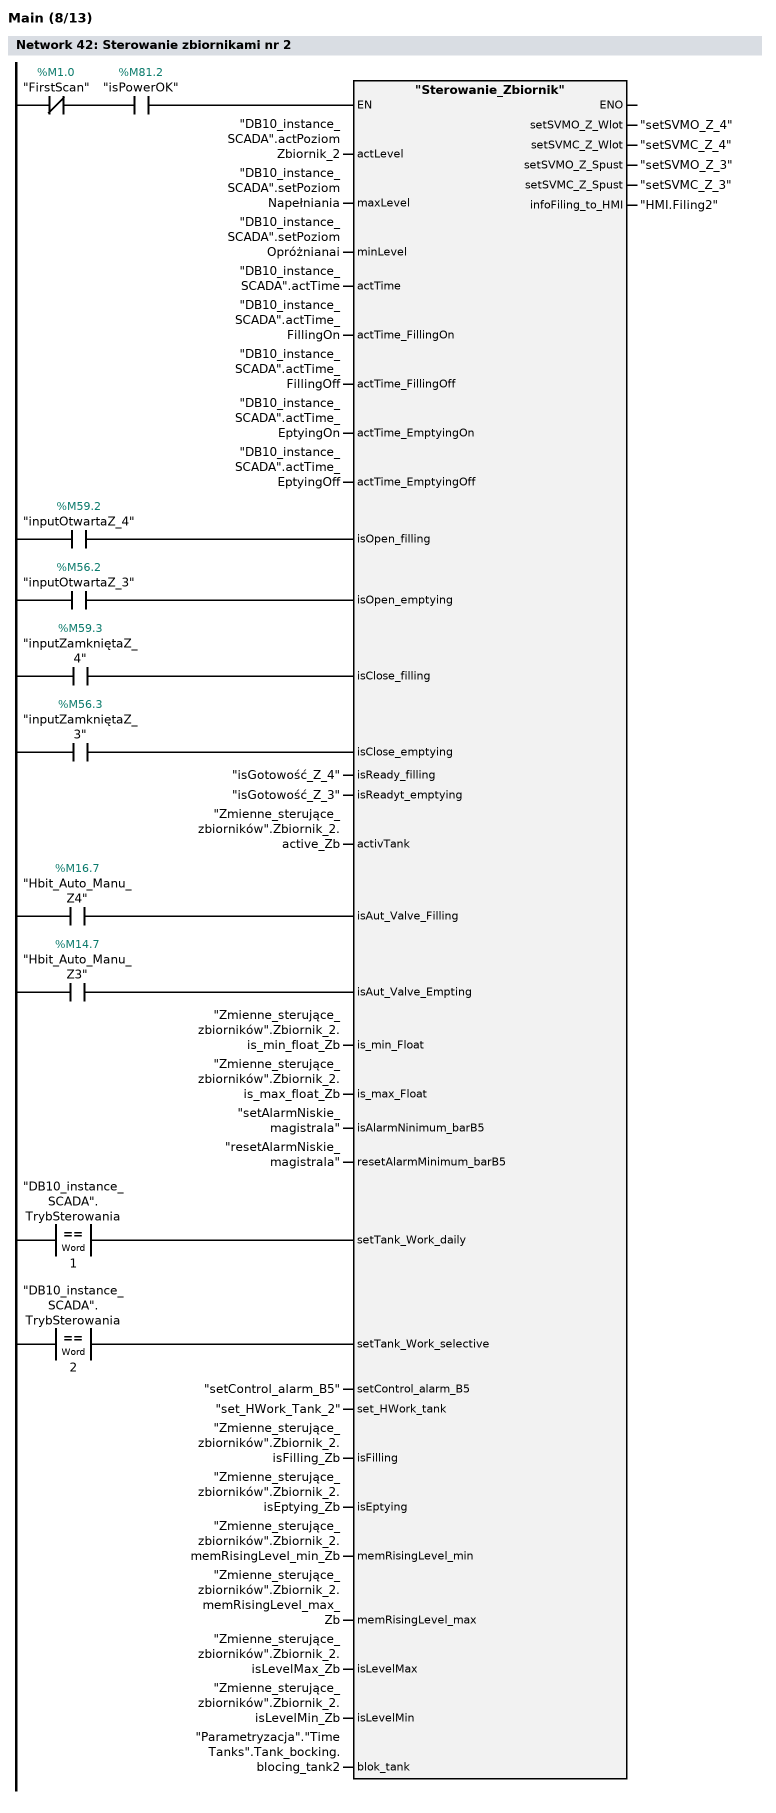
   RUNG wire#powerrail
      I_Contact( "FirstScan" )
      Contact( "isPowerOK" )
      "Sterowanie_Zbiornik"(isOpen_filling := wire#w1, isOpen_emptying := wire#w2, isClose_filling := wire#w3, isClose_emptying := wire#w4, isAut_Valve_Filling := wire#w5, isAut_Valve_Empting := wire#w6, setTank_Work_daily := wire#w7, setTank_Work_selective := wire#w8, actLevel := "DB10_instance_SCADA".actPoziomZbiornik_2, maxLevel := "DB10_instance_SCADA".setPoziomNapełniania, minLevel := "DB10_instance_SCADA".setPoziomOpróżnianai, actTime := "DB10_instance_SCADA".actTime, actTime_FillingOn := "DB10_instance_SCADA".actTime_FillingOn, actTime_FillingOff := "DB10_instance_SCADA".actTime_FillingOff, actTime_EmptyingOn := "DB10_instance_SCADA".actTime_EptyingOn, actTime_EmptyingOff := "DB10_instance_SCADA".actTime_EptyingOff, isReady_filling := "isGotowość_Z_4", isReadyt_emptying := "isGotowość_Z_3", activTank := "Zmienne_sterujące_zbiorników".Zbiornik_2.active_Zb, is_min_Float := "Zmienne_sterujące_zbiorników".Zbiornik_2.is_min_float_Zb, is_max_Float := "Zmienne_sterujące_zbiorników".Zbiornik_2.is_max_float_Zb, isAlarmNinimum_barB5 := "setAlarmNiskie_magistrala", resetAlarmMinimum_barB5 := "resetAlarmNiskie_magistrala", setControl_alarm_B5 := "setControl_alarm_B5", set_HWork_tank := "set_HWork_Tank_2", isFilling := "Zmienne_sterujące_zbiorników".Zbiornik_2.isFilling_Zb, isEptying := "Zmienne_sterujące_zbiorników".Zbiornik_2.isEptying_Zb, memRisingLevel_min := "Zmienne_sterujące_zbiorników".Zbiornik_2.memRisingLevel_min_Zb, memRisingLevel_max := "Zmienne_sterujące_zbiorników".Zbiornik_2.memRisingLevel_max_Zb, isLevelMax := "Zmienne_sterujące_zbiorników".Zbiornik_2.isLevelMax_Zb, isLevelMin := "Zmienne_sterujące_zbiorników".Zbiornik_2.isLevelMin_Zb, blok_tank := "Parametryzacja"."Time Tanks".Tank_bocking.blocing_tank2, setSVMO_Z_Wlot => "setSVMO_Z_4", setSVMC_Z_Wlot => "setSVMC_Z_4", setSVMO_Z_Spust => "setSVMO_Z_3", setSVMC_Z_Spust => "setSVMC_Z_3", infoFiling_to_HMI => "HMI.Filing2")
   END_RUNG
   RUNG wire#powerrail
      Contact( "inputOtwartaZ_4" )
   END_RUNG wire#w1
   RUNG wire#powerrail
      Contact( "inputOtwartaZ_3" )
   END_RUNG wire#w2
   RUNG wire#powerrail
      Contact( "inputZamkniętaZ_4" )
   END_RUNG wire#w3
   RUNG wire#powerrail
      Contact( "inputZamkniętaZ_3" )
   END_RUNG wire#w4
   RUNG wire#powerrail
      Contact( "Hbit_Auto_Manu_Z4" )
   END_RUNG wire#w5
   RUNG wire#powerrail
      Contact( "Hbit_Auto_Manu_Z3" )
   END_RUNG wire#w6
   RUNG wire#powerrail
      { S7_Templates := "SrcType := Word" } EQ_Contact(in1 := "DB10_instance_SCADA".TrybSterowania, in2 := 1)
   END_RUNG wire#w7
   RUNG wire#powerrail
      { S7_Templates := "SrcType := Word" } EQ_Contact(in1 := "DB10_instance_SCADA".TrybSterowania, in2 := 2)
   END_RUNG wire#w8
   // the same network as SCL:
   IF NOT "FirstScan" AND "isPowerOK" THEN
       "Sterowanie_Zbiornik"(actLevel := "DB10_instance_SCADA".actPoziomZbiornik_2,
                             maxLevel := "DB10_instance_SCADA".setPoziomNapełniania,
                             minLevel := "DB10_instance_SCADA".setPoziomOpróżnianai,
                             actTime := "DB10_instance_SCADA".actTime,
                             actTime_FillingOn := "DB10_instance_SCADA".actTime_FillingOn,
                             actTime_FillingOff := "DB10_instance_SCADA".actTime_FillingOff,
                             actTime_EmptyingOn := "DB10_instance_SCADA".actTime_EptyingOn,
                             actTime_EmptyingOff := "DB10_instance_SCADA".actTime_EptyingOff,
                             isOpen_filling := "inputOtwartaZ_4",
                             isOpen_emptying := "inputOtwartaZ_3",
                             isClose_filling := "inputZamkniętaZ_4",
                             isClose_emptying := "inputZamkniętaZ_3",
                             isReady_filling := "isGotowość_Z_4",
                             isReadyt_emptying := "isGotowość_Z_3",
                             activTank := "Zmienne_sterujące_zbiorników".Zbiornik_2.active_Zb,
                             isAut_Valve_Filling := "Hbit_Auto_Manu_Z4",
                             isAut_Valve_Empting := "Hbit_Auto_Manu_Z3",
                             is_min_Float := "Zmienne_sterujące_zbiorników".Zbiornik_2.is_min_float_Zb,
                             is_max_Float := "Zmienne_sterujące_zbiorników".Zbiornik_2.is_max_float_Zb,
                             isAlarmNinimum_barB5 := "setAlarmNiskie_magistrala",
                             resetAlarmMinimum_barB5 := "resetAlarmNiskie_magistrala",
                             setTank_Work_daily := "DB10_instance_SCADA".TrybSterowania = 1,
                             setTank_Work_selective := "DB10_instance_SCADA".TrybSterowania = 2,
                             setControl_alarm_B5 := "setControl_alarm_B5",
                             set_HWork_tank := "set_HWork_Tank_2",
                             isFilling := "Zmienne_sterujące_zbiorników".Zbiornik_2.isFilling_Zb,
                             isEptying := "Zmienne_sterujące_zbiorników".Zbiornik_2.isEptying_Zb,
                             memRisingLevel_min := "Zmienne_sterujące_zbiorników".Zbiornik_2.memRisingLevel_min_Zb,
                             memRisingLevel_max := "Zmienne_sterujące_zbiorników".Zbiornik_2.memRisingLevel_max_Zb,
                             isLevelMax := "Zmienne_sterujące_zbiorników".Zbiornik_2.isLevelMax_Zb,
                             isLevelMin := "Zmienne_sterujące_zbiorników".Zbiornik_2.isLevelMin_Zb,
                             blok_tank := "Parametryzacja"."Time Tanks".Tank_bocking.blocing_tank2,
                             setSVMO_Z_Wlot => "setSVMO_Z_4",
                             setSVMC_Z_Wlot => "setSVMC_Z_4",
                             setSVMO_Z_Spust => "setSVMO_Z_3",
                             setSVMC_Z_Spust => "setSVMC_Z_3",
                             infoFiling_to_HMI => "HMI.Filing2");
   END_IF;
END_REGION

REGION Network 43: Sterowanie zbiornikami nr 3
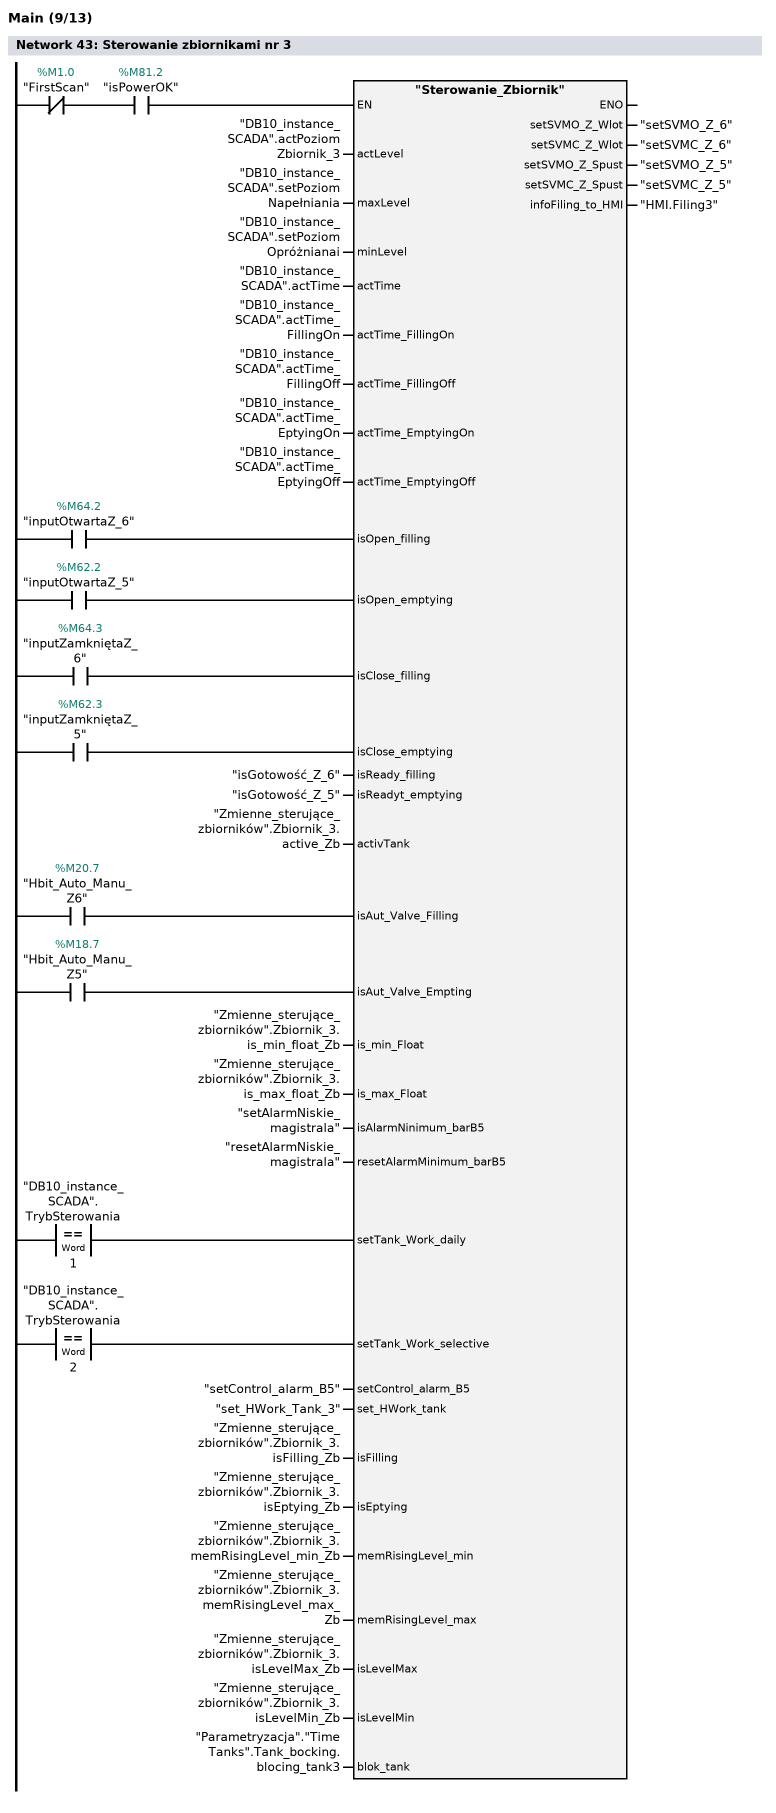
   RUNG wire#powerrail
      I_Contact( "FirstScan" )
      Contact( "isPowerOK" )
      "Sterowanie_Zbiornik"(isOpen_filling := wire#w1, isOpen_emptying := wire#w2, isClose_filling := wire#w3, isClose_emptying := wire#w4, isAut_Valve_Filling := wire#w5, isAut_Valve_Empting := wire#w6, setTank_Work_daily := wire#w7, setTank_Work_selective := wire#w8, actLevel := "DB10_instance_SCADA".actPoziomZbiornik_3, maxLevel := "DB10_instance_SCADA".setPoziomNapełniania, minLevel := "DB10_instance_SCADA".setPoziomOpróżnianai, actTime := "DB10_instance_SCADA".actTime, actTime_FillingOn := "DB10_instance_SCADA".actTime_FillingOn, actTime_FillingOff := "DB10_instance_SCADA".actTime_FillingOff, actTime_EmptyingOn := "DB10_instance_SCADA".actTime_EptyingOn, actTime_EmptyingOff := "DB10_instance_SCADA".actTime_EptyingOff, isReady_filling := "isGotowość_Z_6", isReadyt_emptying := "isGotowość_Z_5", activTank := "Zmienne_sterujące_zbiorników".Zbiornik_3.active_Zb, is_min_Float := "Zmienne_sterujące_zbiorników".Zbiornik_3.is_min_float_Zb, is_max_Float := "Zmienne_sterujące_zbiorników".Zbiornik_3.is_max_float_Zb, isAlarmNinimum_barB5 := "setAlarmNiskie_magistrala", resetAlarmMinimum_barB5 := "resetAlarmNiskie_magistrala", setControl_alarm_B5 := "setControl_alarm_B5", set_HWork_tank := "set_HWork_Tank_3", isFilling := "Zmienne_sterujące_zbiorników".Zbiornik_3.isFilling_Zb, isEptying := "Zmienne_sterujące_zbiorników".Zbiornik_3.isEptying_Zb, memRisingLevel_min := "Zmienne_sterujące_zbiorników".Zbiornik_3.memRisingLevel_min_Zb, memRisingLevel_max := "Zmienne_sterujące_zbiorników".Zbiornik_3.memRisingLevel_max_Zb, isLevelMax := "Zmienne_sterujące_zbiorników".Zbiornik_3.isLevelMax_Zb, isLevelMin := "Zmienne_sterujące_zbiorników".Zbiornik_3.isLevelMin_Zb, blok_tank := "Parametryzacja"."Time Tanks".Tank_bocking.blocing_tank3, setSVMO_Z_Wlot => "setSVMO_Z_6", setSVMC_Z_Wlot => "setSVMC_Z_6", setSVMO_Z_Spust => "setSVMO_Z_5", setSVMC_Z_Spust => "setSVMC_Z_5", infoFiling_to_HMI => "HMI.Filing3")
   END_RUNG
   RUNG wire#powerrail
      Contact( "inputOtwartaZ_6" )
   END_RUNG wire#w1
   RUNG wire#powerrail
      Contact( "inputOtwartaZ_5" )
   END_RUNG wire#w2
   RUNG wire#powerrail
      Contact( "inputZamkniętaZ_6" )
   END_RUNG wire#w3
   RUNG wire#powerrail
      Contact( "inputZamkniętaZ_5" )
   END_RUNG wire#w4
   RUNG wire#powerrail
      Contact( "Hbit_Auto_Manu_Z6" )
   END_RUNG wire#w5
   RUNG wire#powerrail
      Contact( "Hbit_Auto_Manu_Z5" )
   END_RUNG wire#w6
   RUNG wire#powerrail
      { S7_Templates := "SrcType := Word" } EQ_Contact(in1 := "DB10_instance_SCADA".TrybSterowania, in2 := 1)
   END_RUNG wire#w7
   RUNG wire#powerrail
      { S7_Templates := "SrcType := Word" } EQ_Contact(in1 := "DB10_instance_SCADA".TrybSterowania, in2 := 2)
   END_RUNG wire#w8
   // the same network as SCL:
   IF NOT "FirstScan" AND "isPowerOK" THEN
       "Sterowanie_Zbiornik"(actLevel := "DB10_instance_SCADA".actPoziomZbiornik_3,
                             maxLevel := "DB10_instance_SCADA".setPoziomNapełniania,
                             minLevel := "DB10_instance_SCADA".setPoziomOpróżnianai,
                             actTime := "DB10_instance_SCADA".actTime,
                             actTime_FillingOn := "DB10_instance_SCADA".actTime_FillingOn,
                             actTime_FillingOff := "DB10_instance_SCADA".actTime_FillingOff,
                             actTime_EmptyingOn := "DB10_instance_SCADA".actTime_EptyingOn,
                             actTime_EmptyingOff := "DB10_instance_SCADA".actTime_EptyingOff,
                             isOpen_filling := "inputOtwartaZ_6",
                             isOpen_emptying := "inputOtwartaZ_5",
                             isClose_filling := "inputZamkniętaZ_6",
                             isClose_emptying := "inputZamkniętaZ_5",
                             isReady_filling := "isGotowość_Z_6",
                             isReadyt_emptying := "isGotowość_Z_5",
                             activTank := "Zmienne_sterujące_zbiorników".Zbiornik_3.active_Zb,
                             isAut_Valve_Filling := "Hbit_Auto_Manu_Z6",
                             isAut_Valve_Empting := "Hbit_Auto_Manu_Z5",
                             is_min_Float := "Zmienne_sterujące_zbiorników".Zbiornik_3.is_min_float_Zb,
                             is_max_Float := "Zmienne_sterujące_zbiorników".Zbiornik_3.is_max_float_Zb,
                             isAlarmNinimum_barB5 := "setAlarmNiskie_magistrala",
                             resetAlarmMinimum_barB5 := "resetAlarmNiskie_magistrala",
                             setTank_Work_daily := "DB10_instance_SCADA".TrybSterowania = 1,
                             setTank_Work_selective := "DB10_instance_SCADA".TrybSterowania = 2,
                             setControl_alarm_B5 := "setControl_alarm_B5",
                             set_HWork_tank := "set_HWork_Tank_3",
                             isFilling := "Zmienne_sterujące_zbiorników".Zbiornik_3.isFilling_Zb,
                             isEptying := "Zmienne_sterujące_zbiorników".Zbiornik_3.isEptying_Zb,
                             memRisingLevel_min := "Zmienne_sterujące_zbiorników".Zbiornik_3.memRisingLevel_min_Zb,
                             memRisingLevel_max := "Zmienne_sterujące_zbiorników".Zbiornik_3.memRisingLevel_max_Zb,
                             isLevelMax := "Zmienne_sterujące_zbiorników".Zbiornik_3.isLevelMax_Zb,
                             isLevelMin := "Zmienne_sterujące_zbiorników".Zbiornik_3.isLevelMin_Zb,
                             blok_tank := "Parametryzacja"."Time Tanks".Tank_bocking.blocing_tank3,
                             setSVMO_Z_Wlot => "setSVMO_Z_6",
                             setSVMC_Z_Wlot => "setSVMC_Z_6",
                             setSVMO_Z_Spust => "setSVMO_Z_5",
                             setSVMC_Z_Spust => "setSVMC_Z_5",
                             infoFiling_to_HMI => "HMI.Filing3");
   END_IF;
END_REGION

REGION Network 44: Sterowanie zbiornikami nr 4
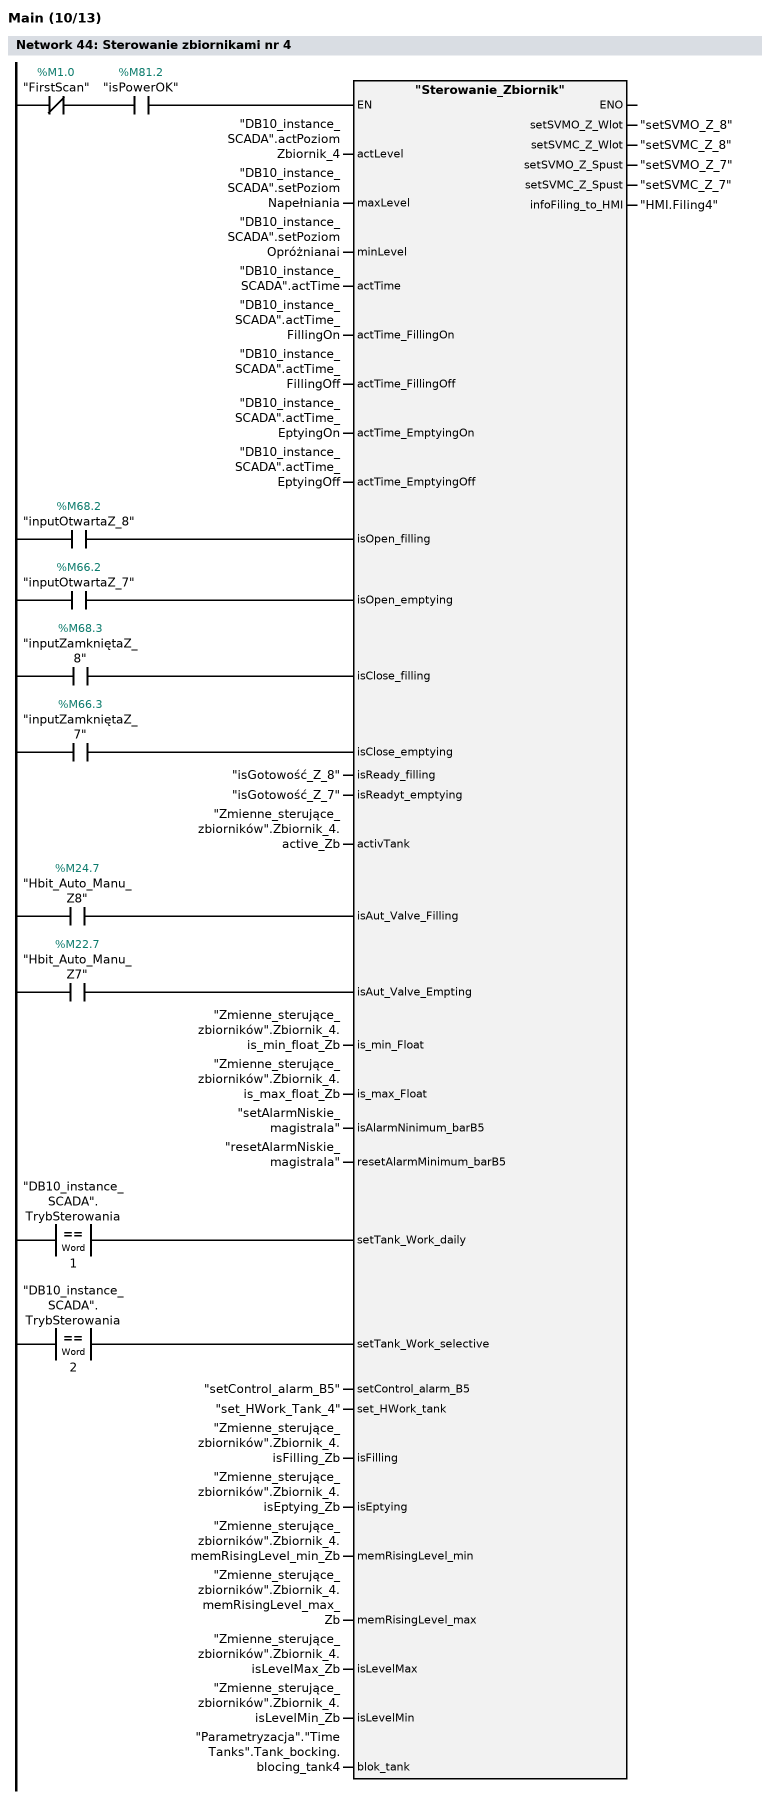
   RUNG wire#powerrail
      I_Contact( "FirstScan" )
      Contact( "isPowerOK" )
      "Sterowanie_Zbiornik"(isOpen_filling := wire#w1, isOpen_emptying := wire#w2, isClose_filling := wire#w3, isClose_emptying := wire#w4, isAut_Valve_Filling := wire#w5, isAut_Valve_Empting := wire#w6, setTank_Work_daily := wire#w7, setTank_Work_selective := wire#w8, actLevel := "DB10_instance_SCADA".actPoziomZbiornik_4, maxLevel := "DB10_instance_SCADA".setPoziomNapełniania, minLevel := "DB10_instance_SCADA".setPoziomOpróżnianai, actTime := "DB10_instance_SCADA".actTime, actTime_FillingOn := "DB10_instance_SCADA".actTime_FillingOn, actTime_FillingOff := "DB10_instance_SCADA".actTime_FillingOff, actTime_EmptyingOn := "DB10_instance_SCADA".actTime_EptyingOn, actTime_EmptyingOff := "DB10_instance_SCADA".actTime_EptyingOff, isReady_filling := "isGotowość_Z_8", isReadyt_emptying := "isGotowość_Z_7", activTank := "Zmienne_sterujące_zbiorników".Zbiornik_4.active_Zb, is_min_Float := "Zmienne_sterujące_zbiorników".Zbiornik_4.is_min_float_Zb, is_max_Float := "Zmienne_sterujące_zbiorników".Zbiornik_4.is_max_float_Zb, isAlarmNinimum_barB5 := "setAlarmNiskie_magistrala", resetAlarmMinimum_barB5 := "resetAlarmNiskie_magistrala", setControl_alarm_B5 := "setControl_alarm_B5", set_HWork_tank := "set_HWork_Tank_4", isFilling := "Zmienne_sterujące_zbiorników".Zbiornik_4.isFilling_Zb, isEptying := "Zmienne_sterujące_zbiorników".Zbiornik_4.isEptying_Zb, memRisingLevel_min := "Zmienne_sterujące_zbiorników".Zbiornik_4.memRisingLevel_min_Zb, memRisingLevel_max := "Zmienne_sterujące_zbiorników".Zbiornik_4.memRisingLevel_max_Zb, isLevelMax := "Zmienne_sterujące_zbiorników".Zbiornik_4.isLevelMax_Zb, isLevelMin := "Zmienne_sterujące_zbiorników".Zbiornik_4.isLevelMin_Zb, blok_tank := "Parametryzacja"."Time Tanks".Tank_bocking.blocing_tank4, setSVMO_Z_Wlot => "setSVMO_Z_8", setSVMC_Z_Wlot => "setSVMC_Z_8", setSVMO_Z_Spust => "setSVMO_Z_7", setSVMC_Z_Spust => "setSVMC_Z_7", infoFiling_to_HMI => "HMI.Filing4")
   END_RUNG
   RUNG wire#powerrail
      Contact( "inputOtwartaZ_8" )
   END_RUNG wire#w1
   RUNG wire#powerrail
      Contact( "inputOtwartaZ_7" )
   END_RUNG wire#w2
   RUNG wire#powerrail
      Contact( "inputZamkniętaZ_8" )
   END_RUNG wire#w3
   RUNG wire#powerrail
      Contact( "inputZamkniętaZ_7" )
   END_RUNG wire#w4
   RUNG wire#powerrail
      Contact( "Hbit_Auto_Manu_Z8" )
   END_RUNG wire#w5
   RUNG wire#powerrail
      Contact( "Hbit_Auto_Manu_Z7" )
   END_RUNG wire#w6
   RUNG wire#powerrail
      { S7_Templates := "SrcType := Word" } EQ_Contact(in1 := "DB10_instance_SCADA".TrybSterowania, in2 := 1)
   END_RUNG wire#w7
   RUNG wire#powerrail
      { S7_Templates := "SrcType := Word" } EQ_Contact(in1 := "DB10_instance_SCADA".TrybSterowania, in2 := 2)
   END_RUNG wire#w8
   // the same network as SCL:
   IF NOT "FirstScan" AND "isPowerOK" THEN
       "Sterowanie_Zbiornik"(actLevel := "DB10_instance_SCADA".actPoziomZbiornik_4,
                             maxLevel := "DB10_instance_SCADA".setPoziomNapełniania,
                             minLevel := "DB10_instance_SCADA".setPoziomOpróżnianai,
                             actTime := "DB10_instance_SCADA".actTime,
                             actTime_FillingOn := "DB10_instance_SCADA".actTime_FillingOn,
                             actTime_FillingOff := "DB10_instance_SCADA".actTime_FillingOff,
                             actTime_EmptyingOn := "DB10_instance_SCADA".actTime_EptyingOn,
                             actTime_EmptyingOff := "DB10_instance_SCADA".actTime_EptyingOff,
                             isOpen_filling := "inputOtwartaZ_8",
                             isOpen_emptying := "inputOtwartaZ_7",
                             isClose_filling := "inputZamkniętaZ_8",
                             isClose_emptying := "inputZamkniętaZ_7",
                             isReady_filling := "isGotowość_Z_8",
                             isReadyt_emptying := "isGotowość_Z_7",
                             activTank := "Zmienne_sterujące_zbiorników".Zbiornik_4.active_Zb,
                             isAut_Valve_Filling := "Hbit_Auto_Manu_Z8",
                             isAut_Valve_Empting := "Hbit_Auto_Manu_Z7",
                             is_min_Float := "Zmienne_sterujące_zbiorników".Zbiornik_4.is_min_float_Zb,
                             is_max_Float := "Zmienne_sterujące_zbiorników".Zbiornik_4.is_max_float_Zb,
                             isAlarmNinimum_barB5 := "setAlarmNiskie_magistrala",
                             resetAlarmMinimum_barB5 := "resetAlarmNiskie_magistrala",
                             setTank_Work_daily := "DB10_instance_SCADA".TrybSterowania = 1,
                             setTank_Work_selective := "DB10_instance_SCADA".TrybSterowania = 2,
                             setControl_alarm_B5 := "setControl_alarm_B5",
                             set_HWork_tank := "set_HWork_Tank_4",
                             isFilling := "Zmienne_sterujące_zbiorników".Zbiornik_4.isFilling_Zb,
                             isEptying := "Zmienne_sterujące_zbiorników".Zbiornik_4.isEptying_Zb,
                             memRisingLevel_min := "Zmienne_sterujące_zbiorników".Zbiornik_4.memRisingLevel_min_Zb,
                             memRisingLevel_max := "Zmienne_sterujące_zbiorników".Zbiornik_4.memRisingLevel_max_Zb,
                             isLevelMax := "Zmienne_sterujące_zbiorników".Zbiornik_4.isLevelMax_Zb,
                             isLevelMin := "Zmienne_sterujące_zbiorników".Zbiornik_4.isLevelMin_Zb,
                             blok_tank := "Parametryzacja"."Time Tanks".Tank_bocking.blocing_tank4,
                             setSVMO_Z_Wlot => "setSVMO_Z_8",
                             setSVMC_Z_Wlot => "setSVMC_Z_8",
                             setSVMO_Z_Spust => "setSVMO_Z_7",
                             setSVMC_Z_Spust => "setSVMC_Z_7",
                             infoFiling_to_HMI => "HMI.Filing4");
   END_IF;
END_REGION

REGION Network 45: Sterowanie zasuwą Z9 odpływu do pompowni
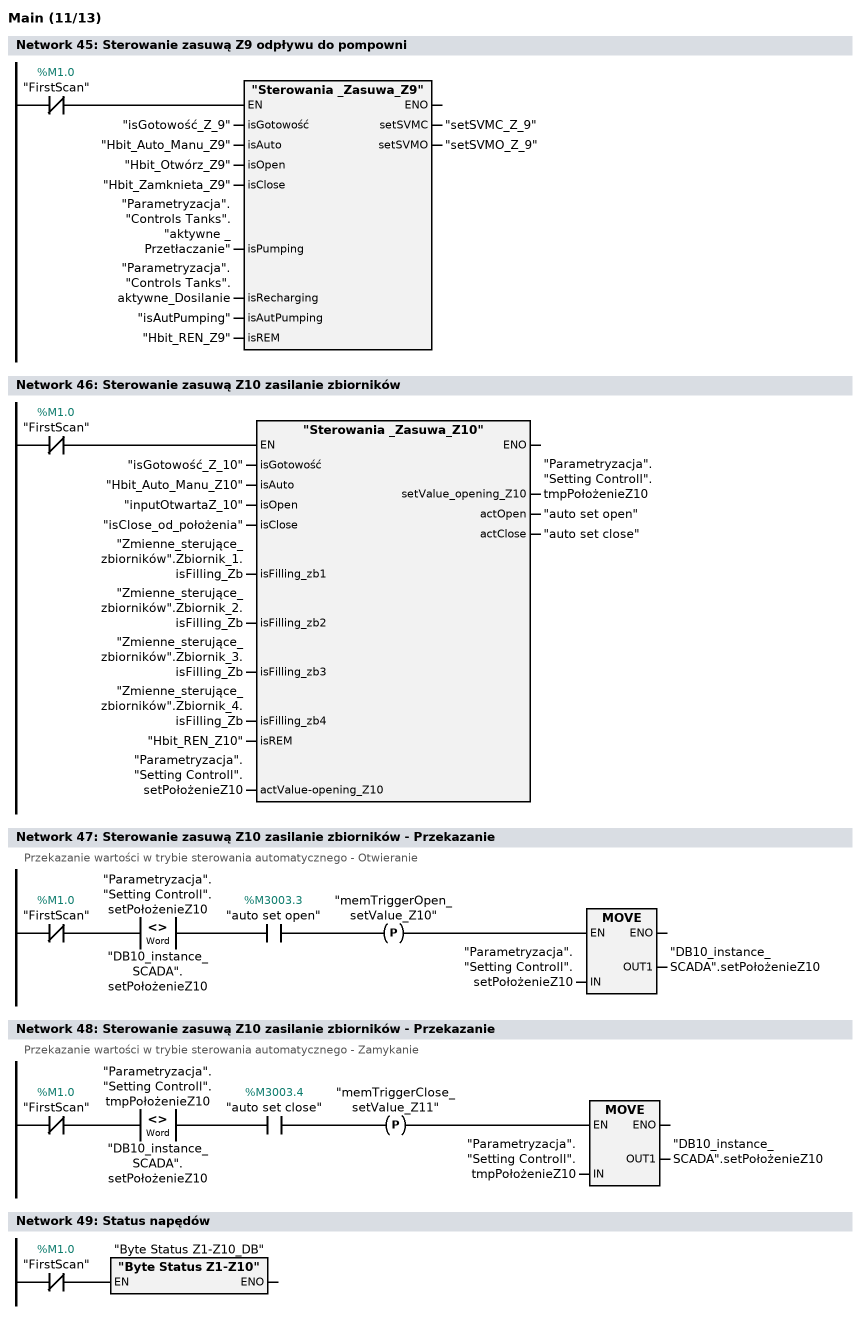
   RUNG wire#powerrail
      I_Contact( "FirstScan" )
      "Sterowania _Zasuwa_Z9"(isGotowość := "isGotowość_Z_9", isAuto := "Hbit_Auto_Manu_Z9", isOpen := "Hbit_Otwórz_Z9", isClose := "Hbit_Zamknieta_Z9", isPumping := "Parametryzacja"."Controls Tanks"."aktywne _Przetłaczanie", isRecharging := "Parametryzacja"."Controls Tanks".aktywne_Dosilanie, isAutPumping := "isAutPumping", isREM := "Hbit_REN_Z9", setSVMC => "setSVMC_Z_9", setSVMO => "setSVMO_Z_9")
   END_RUNG
   // the same network as SCL:
   IF NOT "FirstScan" THEN
       "Sterowania _Zasuwa_Z9"(isGotowość := "isGotowość_Z_9",
                               isAuto := "Hbit_Auto_Manu_Z9",
                               isOpen := "Hbit_Otwórz_Z9",
                               isClose := "Hbit_Zamknieta_Z9",
                               isPumping := "Parametryzacja"."Controls Tanks"."aktywne _Przetłaczanie",
                               isRecharging := "Parametryzacja"."Controls Tanks".aktywne_Dosilanie,
                               isAutPumping := "isAutPumping",
                               isREM := "Hbit_REN_Z9",
                               setSVMC => "setSVMC_Z_9",
                               setSVMO => "setSVMO_Z_9");
   END_IF;
END_REGION

REGION Network 46: Sterowanie zasuwą Z10 zasilanie zbiorników
   RUNG wire#powerrail
      I_Contact( "FirstScan" )
      "Sterowania _Zasuwa_Z10"(isGotowość := "isGotowość_Z_10", isAuto := "Hbit_Auto_Manu_Z10", isOpen := "inputOtwartaZ_10", isClose := "isClose_od_położenia", isFilling_zb1 := "Zmienne_sterujące_zbiorników".Zbiornik_1.isFilling_Zb, isFilling_zb2 := "Zmienne_sterujące_zbiorników".Zbiornik_2.isFilling_Zb, isFilling_zb3 := "Zmienne_sterujące_zbiorników".Zbiornik_3.isFilling_Zb, isFilling_zb4 := "Zmienne_sterujące_zbiorników".Zbiornik_4.isFilling_Zb, isREM := "Hbit_REN_Z10", "actValue-opening_Z10" := "Parametryzacja"."Setting Controll".setPołożenieZ10, setValue_opening_Z10 => "Parametryzacja"."Setting Controll".tmpPołożenieZ10, actOpen => "auto set open", actClose => "auto set close")
   END_RUNG
   // the same network as SCL:
   IF NOT "FirstScan" THEN
       "Sterowania _Zasuwa_Z10"(isGotowość := "isGotowość_Z_10",
                               isAuto := "Hbit_Auto_Manu_Z10",
                               isOpen := "inputOtwartaZ_10",
                               isClose := "isClose_od_położenia",
                               isFilling_zb1 := "Zmienne_sterujące_zbiorników".Zbiornik_1.isFilling_Zb,
                               isFilling_zb2 := "Zmienne_sterujące_zbiorników".Zbiornik_2.isFilling_Zb,
                               isFilling_zb3 := "Zmienne_sterujące_zbiorników".Zbiornik_3.isFilling_Zb,
                               isFilling_zb4 := "Zmienne_sterujące_zbiorników".Zbiornik_4.isFilling_Zb,
                               isREM := "Hbit_REN_Z10",
                               "actValue-opening_Z10" := "Parametryzacja"."Setting Controll".setPołożenieZ10,
                               setValue_opening_Z10 => "Parametryzacja"."Setting Controll".tmpPołożenieZ10,
                               actOpen => "auto set open",
                               actClose => "auto set close");
   END_IF;
END_REGION

REGION Network 47: Sterowanie zasuwą Z10 zasilanie zbiorników - Przekazanie
   // Przekazanie wartości w trybie sterowania automatycznego - Otwieranie
   RUNG wire#powerrail
      I_Contact( "FirstScan" )
      { S7_Templates := "SrcType := Word" } NE_Contact(in1 := "Parametryzacja"."Setting Controll".setPołożenieZ10, in2 := "DB10_instance_SCADA".setPołożenieZ10)
      Contact( "auto set open" )
      P_Trig( "memTriggerOpen_setValue_Z10" )
      Move(in := "Parametryzacja"."Setting Controll".setPołożenieZ10, out1 => "DB10_instance_SCADA".setPołożenieZ10)
   END_RUNG
   // the same network as SCL:
   #_w1 := NOT "FirstScan" AND ("Parametryzacja"."Setting Controll".setPołożenieZ10 <> "DB10_instance_SCADA".setPołożenieZ10) AND "auto set open";
   #_w2 := #_w1 AND NOT "memTriggerOpen_setValue_Z10";   // rising edge
   "memTriggerOpen_setValue_Z10" := #_w1;
   IF #_w2 THEN
       "DB10_instance_SCADA".setPołożenieZ10 := "Parametryzacja"."Setting Controll".setPołożenieZ10;
   END_IF;
END_REGION

REGION Network 48: Sterowanie zasuwą Z10 zasilanie zbiorników - Przekazanie
   // Przekazanie wartości w trybie sterowania automatycznego - Zamykanie
   RUNG wire#powerrail
      I_Contact( "FirstScan" )
      { S7_Templates := "SrcType := Word" } NE_Contact(in1 := "Parametryzacja"."Setting Controll".tmpPołożenieZ10, in2 := "DB10_instance_SCADA".setPołożenieZ10)
      Contact( "auto set close" )
      P_Trig( "memTriggerClose_setValue_Z11" )
      Move(in := "Parametryzacja"."Setting Controll".tmpPołożenieZ10, out1 => "DB10_instance_SCADA".setPołożenieZ10)
   END_RUNG
   // the same network as SCL:
   #_w1 := NOT "FirstScan" AND ("Parametryzacja"."Setting Controll".tmpPołożenieZ10 <> "DB10_instance_SCADA".setPołożenieZ10) AND "auto set close";
   #_w2 := #_w1 AND NOT "memTriggerClose_setValue_Z11";   // rising edge
   "memTriggerClose_setValue_Z11" := #_w1;
   IF #_w2 THEN
       "DB10_instance_SCADA".setPołożenieZ10 := "Parametryzacja"."Setting Controll".tmpPołożenieZ10;
   END_IF;
END_REGION

REGION Network 49: Status napędów
   RUNG wire#powerrail
      I_Contact( "FirstScan" )
      "Byte Status Z1-Z10_DB"()
   END_RUNG
   // the same network as SCL:
   IF NOT "FirstScan" THEN
       "Byte Status Z1-Z10_DB"();   // "Byte Status Z1-Z10"
   END_IF;
END_REGION

REGION Network 50: Kontrola styków momentowych
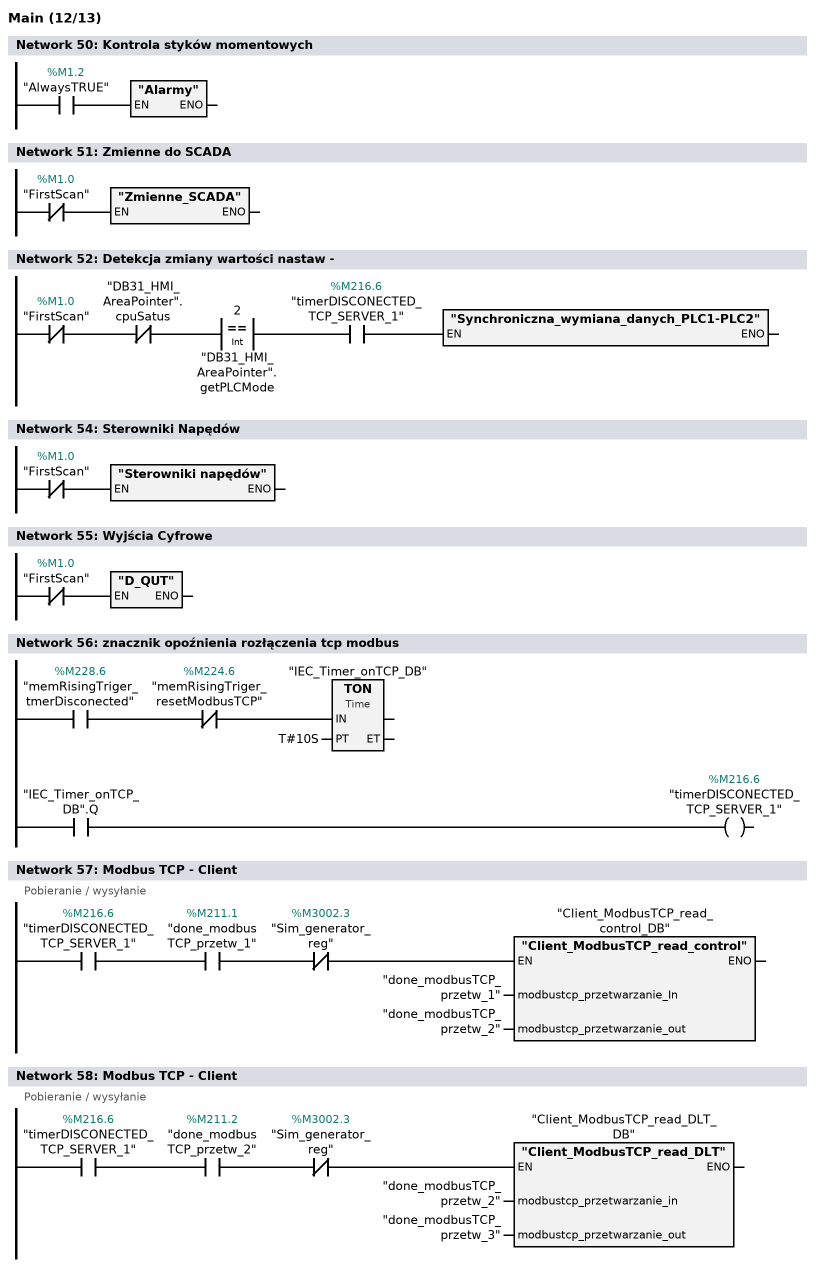
   RUNG wire#powerrail
      Contact( "AlwaysTRUE" )
      "Alarmy"()
   END_RUNG
   // the same network as SCL:
   IF "AlwaysTRUE" THEN "Alarmy"(); END_IF;
END_REGION

REGION Network 51: Zmienne do SCADA
   RUNG wire#powerrail
      I_Contact( "FirstScan" )
      "Zmienne_SCADA"()
   END_RUNG
   // the same network as SCL:
   IF NOT "FirstScan" THEN "Zmienne_SCADA"(); END_IF;
END_REGION

REGION Network 52: Detekcja zmiany wartości nastaw -
   RUNG wire#powerrail
      I_Contact( "FirstScan" )
      I_Contact( "DB31_HMI_AreaPointer".cpuSatus )
      { S7_Templates := "SrcType := Int" } EQ_Contact(in1 := 2, in2 := "DB31_HMI_AreaPointer".getPLCMode)
      Contact( "timerDISCONECTED_TCP_SERVER_1" )
      "Synchroniczna_wymiana_danych_PLC1-PLC2"()
   END_RUNG
   // the same network as SCL:
   IF NOT "FirstScan" AND NOT "DB31_HMI_AreaPointer".cpuSatus AND (2 = "DB31_HMI_AreaPointer".getPLCMode) AND "timerDISCONECTED_TCP_SERVER_1" THEN
       "Synchroniczna_wymiana_danych_PLC1-PLC2"();
   END_IF;
END_REGION

REGION Network 53
   // Funkcja po przeprowadzeniu sprawdzenia czy nastąpiły zmiany w danych przekazuje nowe wartości
END_REGION

REGION Network 54: Sterowniki Napędów
   RUNG wire#powerrail
      I_Contact( "FirstScan" )
      "Sterowniki napędów"()
   END_RUNG
   // the same network as SCL:
   IF NOT "FirstScan" THEN "Sterowniki napędów"(); END_IF;
END_REGION

REGION Network 55: Wyjścia Cyfrowe
   RUNG wire#powerrail
      I_Contact( "FirstScan" )
      "D_QUT"()
   END_RUNG
   // the same network as SCL:
   IF NOT "FirstScan" THEN "D_QUT"(); END_IF;
END_REGION

REGION Network 56: znacznik opoźnienia rozłączenia tcp modbus
   RUNG wire#powerrail
      Contact( "memRisingTriger_tmerDisconected" )
      I_Contact( "memRisingTriger_resetModbusTCP" )
      { S7_Templates := "time_type := Time" } "IEC_Timer_onTCP_DB".TON(pt := T#10S, et =>)
   END_RUNG
   RUNG wire#powerrail
      Contact( "IEC_Timer_onTCP_DB".Q )
      Coil( "timerDISCONECTED_TCP_SERVER_1" )
   END_RUNG
   // the same network as SCL:
   "IEC_Timer_onTCP_DB".TON(IN := "memRisingTriger_tmerDisconected" AND NOT "memRisingTriger_resetModbusTCP",
                           PT := T#10S);
   "timerDISCONECTED_TCP_SERVER_1" := "IEC_Timer_onTCP_DB".Q;
END_REGION

REGION Network 57: Modbus TCP - Client
   // Pobieranie / wysyłanie
   RUNG wire#powerrail
      Contact( "timerDISCONECTED_TCP_SERVER_1" )
      Contact( "done_modbusTCP_przetw_1" )
      I_Contact( "Sim_generator_reg" )
      "Client_ModbusTCP_read_control_DB"(modbustcp_przetwarzanie_In := "done_modbusTCP_przetw_1", modbustcp_przetwarzanie_out := "done_modbusTCP_przetw_2")
   END_RUNG
   // the same network as SCL:
   IF "timerDISCONECTED_TCP_SERVER_1" AND "done_modbusTCP_przetw_1" AND NOT "Sim_generator_reg" THEN
       "Client_ModbusTCP_read_control_DB"(modbustcp_przetwarzanie_In := "done_modbusTCP_przetw_1",   // "Client_ModbusTCP_read_control"
                               modbustcp_przetwarzanie_out := "done_modbusTCP_przetw_2");
   END_IF;
END_REGION

REGION Network 58: Modbus TCP - Client
   // Pobieranie / wysyłanie
   RUNG wire#powerrail
      Contact( "timerDISCONECTED_TCP_SERVER_1" )
      Contact( "done_modbusTCP_przetw_2" )
      I_Contact( "Sim_generator_reg" )
      "Client_ModbusTCP_read_DLT_DB"(modbustcp_przetwarzanie_in := "done_modbusTCP_przetw_2", modbustcp_przetwarzanie_out := "done_modbusTCP_przetw_3")
   END_RUNG
   // the same network as SCL:
   IF "timerDISCONECTED_TCP_SERVER_1" AND "done_modbusTCP_przetw_2" AND NOT "Sim_generator_reg" THEN
       "Client_ModbusTCP_read_DLT_DB"(modbustcp_przetwarzanie_in := "done_modbusTCP_przetw_2",   // "Client_ModbusTCP_read_DLT"
                               modbustcp_przetwarzanie_out := "done_modbusTCP_przetw_3");
   END_IF;
END_REGION

REGION Network 59: Modbus TCP - Client
   // Pobieranie / wysyłanie
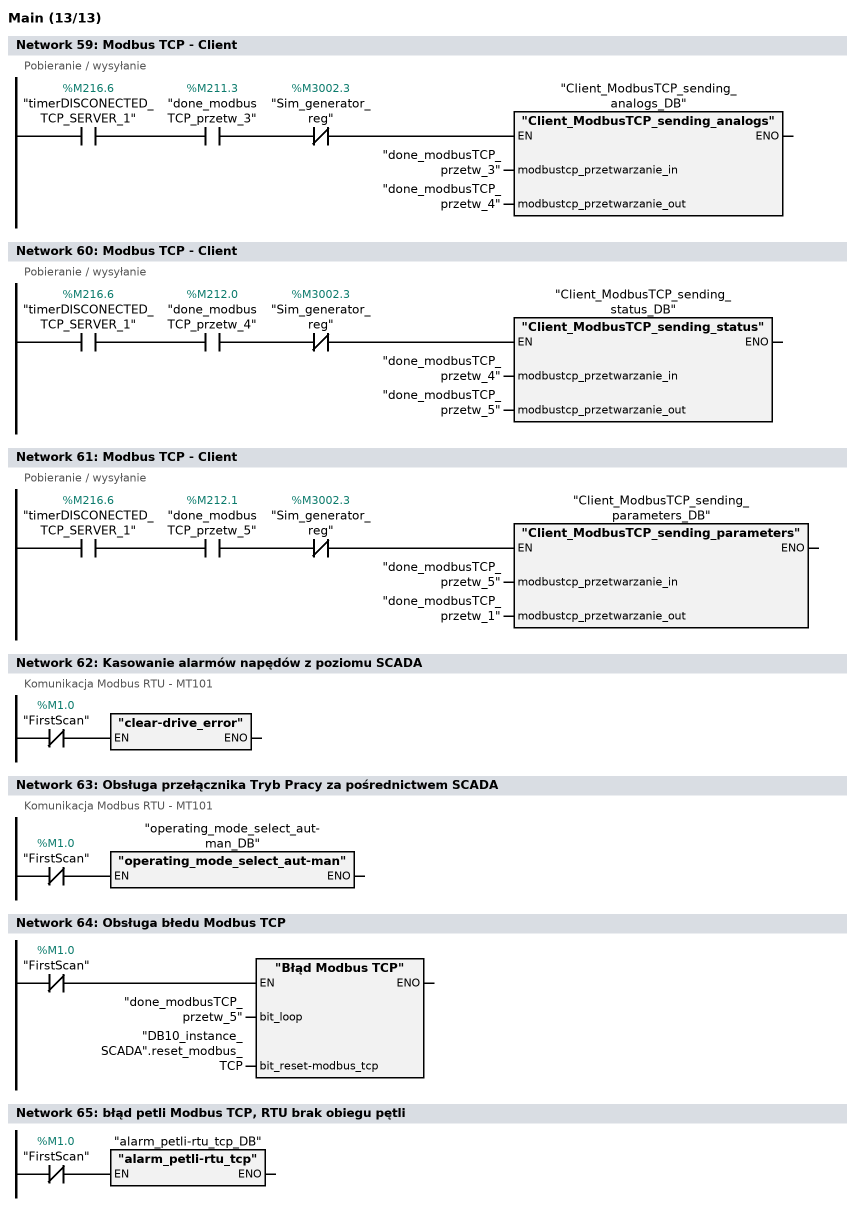
   RUNG wire#powerrail
      Contact( "timerDISCONECTED_TCP_SERVER_1" )
      Contact( "done_modbusTCP_przetw_3" )
      I_Contact( "Sim_generator_reg" )
      "Client_ModbusTCP_sending_analogs_DB"(modbustcp_przetwarzanie_in := "done_modbusTCP_przetw_3", modbustcp_przetwarzanie_out := "done_modbusTCP_przetw_4")
   END_RUNG
   // the same network as SCL:
   IF "timerDISCONECTED_TCP_SERVER_1" AND "done_modbusTCP_przetw_3" AND NOT "Sim_generator_reg" THEN
       "Client_ModbusTCP_sending_analogs_DB"(modbustcp_przetwarzanie_in := "done_modbusTCP_przetw_3",   // "Client_ModbusTCP_sending_analogs"
                               modbustcp_przetwarzanie_out := "done_modbusTCP_przetw_4");
   END_IF;
END_REGION

REGION Network 60: Modbus TCP - Client
   // Pobieranie / wysyłanie
   RUNG wire#powerrail
      Contact( "timerDISCONECTED_TCP_SERVER_1" )
      Contact( "done_modbusTCP_przetw_4" )
      I_Contact( "Sim_generator_reg" )
      "Client_ModbusTCP_sending_status_DB"(modbustcp_przetwarzanie_in := "done_modbusTCP_przetw_4", modbustcp_przetwarzanie_out := "done_modbusTCP_przetw_5")
   END_RUNG
   // the same network as SCL:
   IF "timerDISCONECTED_TCP_SERVER_1" AND "done_modbusTCP_przetw_4" AND NOT "Sim_generator_reg" THEN
       "Client_ModbusTCP_sending_status_DB"(modbustcp_przetwarzanie_in := "done_modbusTCP_przetw_4",   // "Client_ModbusTCP_sending_status"
                               modbustcp_przetwarzanie_out := "done_modbusTCP_przetw_5");
   END_IF;
END_REGION

REGION Network 61: Modbus TCP - Client
   // Pobieranie / wysyłanie
   RUNG wire#powerrail
      Contact( "timerDISCONECTED_TCP_SERVER_1" )
      Contact( "done_modbusTCP_przetw_5" )
      I_Contact( "Sim_generator_reg" )
      "Client_ModbusTCP_sending_parameters_DB"(modbustcp_przetwarzanie_in := "done_modbusTCP_przetw_5", modbustcp_przetwarzanie_out := "done_modbusTCP_przetw_1")
   END_RUNG
   // the same network as SCL:
   IF "timerDISCONECTED_TCP_SERVER_1" AND "done_modbusTCP_przetw_5" AND NOT "Sim_generator_reg" THEN
       "Client_ModbusTCP_sending_parameters_DB"(modbustcp_przetwarzanie_in := "done_modbusTCP_przetw_5",   // "Client_ModbusTCP_sending_parameters"
                               modbustcp_przetwarzanie_out := "done_modbusTCP_przetw_1");
   END_IF;
END_REGION

REGION Network 62: Kasowanie alarmów napędów z poziomu SCADA
   // Komunikacja Modbus RTU - MT101
   RUNG wire#powerrail
      I_Contact( "FirstScan" )
      "clear-drive_error"()
   END_RUNG
   // the same network as SCL:
   IF NOT "FirstScan" THEN "clear-drive_error"(); END_IF;
END_REGION

REGION Network 63: Obsługa przełącznika Tryb Pracy za pośrednictwem SCADA
   // Komunikacja Modbus RTU - MT101
   RUNG wire#powerrail
      I_Contact( "FirstScan" )
      "operating_mode_select_aut-man_DB"()
   END_RUNG
   // the same network as SCL:
   IF NOT "FirstScan" THEN
       "operating_mode_select_aut-man_DB"();   // "operating_mode_select_aut-man"
   END_IF;
END_REGION

REGION Network 64: Obsługa błedu Modbus TCP
   RUNG wire#powerrail
      I_Contact( "FirstScan" )
      "Błąd Modbus TCP"(bit_loop := "done_modbusTCP_przetw_5", "bit_reset-modbus_tcp" := "DB10_instance_SCADA".reset_modbus_TCP)
   END_RUNG
   // the same network as SCL:
   IF NOT "FirstScan" THEN
       "Błąd Modbus TCP"(bit_loop := "done_modbusTCP_przetw_5",
                         "bit_reset-modbus_tcp" := "DB10_instance_SCADA".reset_modbus_TCP);
   END_IF;
END_REGION

REGION Network 65: błąd petli Modbus TCP, RTU brak obiegu pętli
   RUNG wire#powerrail
      I_Contact( "FirstScan" )
      "alarm_petli-rtu_tcp_DB"()
   END_RUNG
   // the same network as SCL:
   IF NOT "FirstScan" THEN
       "alarm_petli-rtu_tcp_DB"();   // "alarm_petli-rtu_tcp"
   END_IF;
END_REGION
END_ORGANIZATION_BLOCK

FUNCTION "Start_upPower" : Void   // FC22, LAD
TITLE = Start po restarcie
{ S7_Optimized_Access := 'TRUE' }
AUTHOR : rtecmer
VERSION : 0.1
// opóznienie aktualizacji stanów gotowości itp.
// stored: AutoNumber true, IsIECCheckEnabled false, SetENOAutomatically false, UDAEnableTagReadback false
   VAR_INPUT
      KT1 : Time;   // Czas timera
   END_VAR
   VAR_IN_OUT
      TMR1 : TON_TIME;
      isPowerOK : Bool;
   END_VAR
BEGIN

REGION Network 1
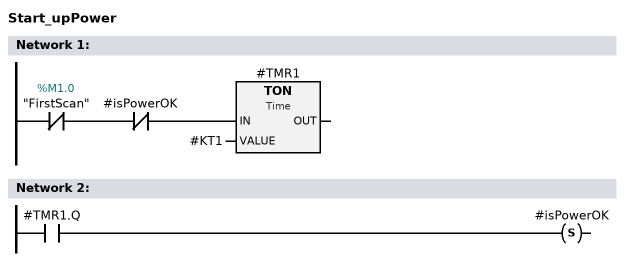
   #TMR1(IN := NOT "FirstScan" AND NOT #isPowerOK, PT := #KT1);   // TON coil
END_REGION

REGION Network 2
   RUNG wire#powerrail
      Contact( #TMR1.Q )
      S_Coil( #isPowerOK )
   END_RUNG
   // the same network as SCL:
   IF #TMR1.Q THEN #isPowerOK := TRUE; END_IF;
END_REGION
END_FUNCTION

FUNCTION "RTC" : Void   // FC44, LAD
{ S7_Optimized_Access := 'TRUE' }
VERSION : 0.1
// stored: AutoNumber true, IsIECCheckEnabled false, SetENOAutomatically false, UDAEnableTagReadback false
   VAR_TEMP   // added for the SCL form of the ladder/FBD networks
      _w1 : Bool;
      _w2 : Bool;
   END_VAR
BEGIN

REGION Network 1
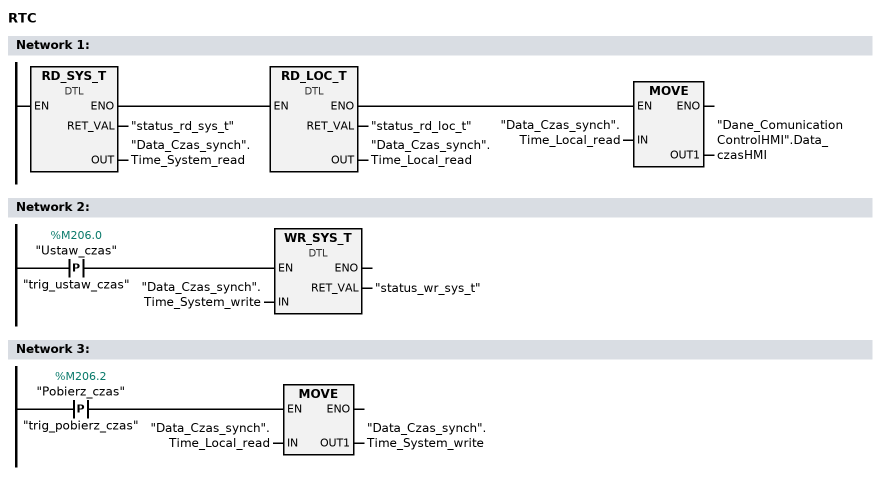
   RUNG wire#powerrail
      { S7_Templates := "date_type := DTL" } RD_SYS_T(RET_VAL => "status_rd_sys_t", OUT => "Data_Czas_synch".Time_System_read)
      { S7_Templates := "date_type := DTL" } RD_LOC_T(RET_VAL => "status_rd_loc_t", OUT => "Data_Czas_synch".Time_Local_read)
      { S7_GenerateENO := "TRUE" } Move(in := "Data_Czas_synch".Time_Local_read, out1 => "Dane_ComunicationControlHMI".Data_czasHMI)
   END_RUNG
   // the same network as SCL:
   "status_rd_sys_t" := RD_SYS_T(OUT => "Data_Czas_synch".Time_System_read, ENO => #_w1);
   "status_rd_loc_t" := RD_LOC_T(EN := #_w1, OUT => "Data_Czas_synch".Time_Local_read, ENO => #_w2);
   IF #_w2 THEN "Dane_ComunicationControlHMI".Data_czasHMI := "Data_Czas_synch".Time_Local_read; END_IF;
END_REGION

REGION Network 2
   RUNG wire#powerrail
      P_Contact(operand := "Ustaw_czas", bit := "trig_ustaw_czas")
      { S7_Templates := "date_type := DTL" } WR_SYS_T(IN := "Data_Czas_synch".Time_System_write, RET_VAL => "status_wr_sys_t")
   END_RUNG
   // the same network as SCL:
   #_w1 := "Ustaw_czas" AND NOT "trig_ustaw_czas";   // rising edge of "Ustaw_czas"
   "trig_ustaw_czas" := "Ustaw_czas";
   IF #_w1 THEN "status_wr_sys_t" := WR_SYS_T(IN := "Data_Czas_synch".Time_System_write); END_IF;
END_REGION

REGION Network 3
   RUNG wire#powerrail
      P_Contact(operand := "Pobierz_czas", bit := "trig_pobierz_czas")
      { S7_GenerateENO := "TRUE" } Move(in := "Data_Czas_synch".Time_Local_read, out1 => "Data_Czas_synch".Time_System_write)
   END_RUNG
   // the same network as SCL:
   #_w1 := "Pobierz_czas" AND NOT "trig_pobierz_czas";   // rising edge of "Pobierz_czas"
   "trig_pobierz_czas" := "Pobierz_czas";
   IF #_w1 THEN "Data_Czas_synch".Time_System_write := "Data_Czas_synch".Time_Local_read; END_IF;
END_REGION
END_FUNCTION

FUNCTION "LD_ReadLedStatus" : Void
{ S7_Optimized_Access := 'TRUE' }
VERSION : 0.1
   VAR_TEMP 
      tempCounter : Int;
   END_VAR


BEGIN
	FOR #tempCounter := 1 TO 6 BY 1 DO
	    "V_LED".LED[#tempCounter] := "HD_LED"(LED := INT_TO_UINT(IN := #tempCounter));
	END_FOR;
END_FUNCTION

FUNCTION "HD_LED" : Int
{ S7_Optimized_Access := 'TRUE' }
AUTHOR : gilewski
FAMILY : HD
VERSION : 0.1
   VAR_INPUT 
      LED : UInt;
   END_VAR


BEGIN
	#HD_LED := LED(LADDR := "Local~Common",
	               LED := #LED);
	
	"ERR_GetSoftwareError"(Error := #HD_LED > 9,
	                       Status := INT_TO_DWORD(#HD_LED),
	                       Buffer := "ERR_ErrorBufferFull".SoftwareError["ERR_Enum".SoftwareError.LED]);
END_FUNCTION

FUNCTION_BLOCK "EX012_ErrorHandling"
{ S7_Optimized_Access := 'TRUE' }
VERSION : 0.1
   VAR_INPUT RETAIN
      LED : Int;
      CounterError : USInt;
   END_VAR

   VAR_OUTPUT 
      RedLED : Bool;
   END_VAR

   VAR 
      tempCounterDiagStatus : USInt;
      tempCounterError : USInt;
   END_VAR

   VAR_TEMP 
      tempLed : Bool;
   END_VAR


BEGIN
	//Function to set the light detection mark led error
	#tempLed := FALSE;
	#tempCounterError := #CounterError;
	//set temporary narker Led
	IF #LED <> 1 THEN
	    #tempLed := TRUE;
	ELSE
	    #tempLed := FALSE;
	END_IF;
	
	
	//Set marker error
	IF (#tempLed = TRUE) THEN
	    #RedLED := TRUE;
	ELSE
	    #RedLED := FALSE;
	END_IF;
	   
	    
	
	
	
END_FUNCTION_BLOCK

FUNCTION "ERR_ClassReset" : Void
{ S7_Optimized_Access := 'TRUE' }
VERSION : 0.1

BEGIN
	//Reset OB error
	IF ("V_ErrorOB".ResetErrorOB = TRUE) THEN
	    "ERR_ResetOB80"();
	    "V_ErrorOB".OB80 := FALSE;
	    "V_ErrorOB".StartUp.LostRetentive := FALSE;
	    "V_ErrorOB".StartUp.LostRTC := FALSE;
	    "V_ErrorOB".ResetErrorOB := FALSE;
	END_IF;
	//Reset Software error
	IF ("V_SoftwareError".ResetErrorSoftware = TRUE) THEN
	    "ERR_ResetGetError"();
	    "ERR_ResetSoftwareError"();
	    "ERR_ErrorBufferFull".CounterDiagStatusUpdate := 0;
	    "V_SoftwareError".DiagnosticBuffer := FALSE;
	    "V_SoftwareError".GetErrorFunction := FALSE;
	    "V_SoftwareError".SoftwareFunctions := FALSE;
	    "V_SoftwareError".ResetErrorSoftware := FALSE;
	END_IF;
END_FUNCTION

FUNCTION "ERR_ResetOB80" : Void
{ S7_Optimized_Access := 'TRUE' }
VERSION : 0.1
   VAR_TEMP 
      tempCounter : Int;
      tempStructure : "stt_ERR_OB80";
   END_VAR


BEGIN
	//structure initialization
	#tempStructure.Counter := 0;
	#tempStructure.Overflow := 0;
	FOR #tempCounter := 0 TO 4 BY 1 DO
	    #tempStructure.OBnr[#tempCounter] := 0;
	END_FOR;
	//Reset buffer
	FOR #tempCounter := 0 TO 5 BY 1 DO
	    "ERR_ErrorOB".OB80[#tempCounter] := #tempStructure;
	END_FOR;
	
	
END_FUNCTION

FUNCTION "ERR_ResetGetError" : Void
{ S7_Optimized_Access := 'TRUE' }
VERSION : 0.1
   VAR_TEMP 
      tempCounter : Int;
      tempStructure : "stt_ERR_GetError";
   END_VAR


BEGIN
	//structure initialization
	#tempStructure.Counter := 0;
	#tempStructure.Overflow := FALSE;
	FOR #tempCounter := 0 TO 4 BY 1 DO
	    #tempStructure.Component[#tempCounter].BlockNumber := 0;
	    #tempStructure.Component[#tempCounter].BlockType := 0;
	    #tempStructure.Component[#tempCounter].MemoryArea := 0;
	    #tempStructure.Component[#tempCounter].NumberDB := 0;
	END_FOR;
	//Reset buffer
	FOR #tempCounter := 0 TO 27 BY 1 DO
	    "ERR_ErrorBufferFull".GetError[#tempCounter] := #tempStructure;
	END_FOR;
	
	
END_FUNCTION

FUNCTION "ERR_ResetSoftwareError" : Void
{ S7_Optimized_Access := 'TRUE' }
VERSION : 0.1
   VAR_TEMP 
      tempCounter : Int;
      tempStructure : "stt_ERR_SoftwareError";
   END_VAR


BEGIN
	//structure initialization
	#tempStructure.Counter := 0;
	#tempStructure.Overflow := FALSE;
	FOR #tempCounter := 0 TO 4 BY 1 DO
	    #tempStructure.Status[#tempCounter] := 0;
	END_FOR;
	//Reset buffer
	FOR #tempCounter := 0 TO 4 BY 1 DO
	    "ERR_ErrorBufferFull".SoftwareError[#tempCounter] := #tempStructure;
	END_FOR;
	
	
END_FUNCTION

FUNCTION "ERR_ClassGetError" : Void
{ S7_Optimized_Access := 'TRUE' }
VERSION : 0.1
   VAR_TEMP 
      tempErrorData : "stt_ERR_ComponentGetError";
      tempNumberErrorID : Int;
      tempSaveToBuffer : Bool;
   END_VAR


BEGIN
	IF ("ERR_ErrorBufferFull".Error.ERROR_ID <> 0) THEN
	    //copy important data 
	    "ERR_GetErrorFromStructure"(ErrorStructure := "ERR_ErrorBufferFull".Error,
	                                ErrorData => #tempErrorData);
	    // search ErrorID
	    #tempNumberErrorID := "ERR_GetErrorID"(ErrorID := "ERR_ErrorBufferFull".Error.ERROR_ID);
	    IF (#tempNumberErrorID < 0) THEN
	        RETURN;//Error ID not exist!
	    END_IF;
	    // Compare actual component error and component from buffer
	    #tempSaveToBuffer := "ERR_CompareGetErrorComponent"(Actual := #tempErrorData,
	                                                        Buffer := "ERR_ErrorBufferFull".GetError[#tempNumberErrorID]);
	    IF (#tempSaveToBuffer = TRUE) THEN
	        "ERR_OverflowBufferControl"(Counter := "ERR_ErrorBufferFull".GetError[#tempNumberErrorID].Counter,
	                                    Overflow := "ERR_ErrorBufferFull".GetError[#tempNumberErrorID].Overflow);
	        "ERR_SaveErrorToBuffer"(DataToSave := #tempErrorData,
	                                        Buffer := "ERR_ErrorBufferFull".GetError[#tempNumberErrorID]);
	    END_IF;
	END_IF;
	
END_FUNCTION

FUNCTION "ERR_GetErrorFromStructure" : Void
{ S7_Optimized_Access := 'TRUE' }
VERSION : 0.1
   VAR_INPUT 
      ErrorStructure {InstructionName := 'ErrorStruct'; LibVersion := '1.0'} : ErrorStruct;
   END_VAR

   VAR_OUTPUT 
      ErrorData : "stt_ERR_ComponentGetError";
   END_VAR


BEGIN
	#ErrorData.BlockNumber := #ErrorStructure.CODE_ADDRESS.CB_NUMBER;
	#ErrorData.BlockType := #ErrorStructure.CODE_ADDRESS.BLOCK_TYPE;
	#ErrorData.MemoryArea := #ErrorStructure.DATA_ADDRESS.AREA;
	#ErrorData.NumberDB := #ErrorStructure.DATA_ADDRESS.DB_NUMBER;
	
END_FUNCTION

FUNCTION "ERR_GetErrorID" : Int
{ S7_Optimized_Access := 'TRUE' }
VERSION : 0.1
   VAR_INPUT 
      ErrorID : Word;
   END_VAR

   VAR_TEMP 
      tempCounter : Int;
   END_VAR


BEGIN
	#ERR_GetErrorID := -1;
	//searching ID
	FOR #tempCounter := 0 TO 27 BY 1 DO
	    IF (#ErrorID = "ERR_Enum".GetErrorID[#tempCounter]) THEN
	        #ERR_GetErrorID := #tempCounter;
	        RETURN;
	    END_IF;
	END_FOR;
	
END_FUNCTION

FUNCTION "ERR_SaveErrorToBuffer" : Void
{ S7_Optimized_Access := 'TRUE' }
VERSION : 0.1
   VAR_INPUT 
      DataToSave : "stt_ERR_ComponentGetError";
   END_VAR

   VAR_IN_OUT 
      Buffer : "stt_ERR_GetError";
   END_VAR

   VAR_TEMP 
      tempCounter : USInt;
   END_VAR


BEGIN
	//#tempCounter := #PlaceToSave.Counter;
	//#PlaceToSave.Component[#tempCounter] := #DataToSave;   
	#Buffer.Component[#Buffer.Counter] := #DataToSave;
END_FUNCTION

FUNCTION "Wybór_Trybu_Sterowania" : Void
TITLE = Tryb sterowania
{ S7_Optimized_Access := 'TRUE' }
AUTHOR : rtecmer
VERSION : 0.1
//Dostepne tryby sterowania zbiornikami: Wyłączony, Dobowy, Tygodniowy, Ręczny

BEGIN
	(*
	//=============================================================================
	//(JZWiK S.A Radosław Tecmer)
	//(c)Copyright (2022) All Rights Reserved
	//-----------------------------------------------------------------------------
	//Testowane z:   (system docelowy z  FW 4.4)
	//Pakiet inżynierski:   TIA Portal (V16 Update 5)
	//Ograniczenia:  ( - )
	//Wymagania:  (minimalne S7-1200 CPU 1215C FW 4.2 .)
	//Funkcjonalnośc: (Pobranie informacji wybranego trybu sterowania zbiornikami 
	                   i ustawienie znaczników isPumping, isRecharging)
	//-----------------------------------------------------------------------------
	//Zmainy wprowadzone:
	//Wersja  Data       Osoba wprowadzająca zmiany - ekspert
	//01.00.00 02.04.2022 (Tecmer Radosław - twórca) Pieresza wersja 01.00.00
	//=============================================================================
	*)
	
	REGION Detekcja wybranego modelu sterowania pompownią  
	  // 
	  CASE "DB10_instance_SCADA".ModelSterowania OF
	    0:  // Wyłączone
	      "isRecharging" := FALSE;
	      "isPumping" := False;
	      "isAutPumping" := FALSE;
	      
	      ;
	    1:  // Dosilanie
	      "isRecharging" := TRUE;
	      "isPumping" := False;
	      "isAutPumping" := FALSE;
	      ;
	    2: //  Przetłaczanie 
	      "isRecharging" := FALSE;
	      "isPumping" := TRUE;
	      "isAutPumping" := FALSE;
	      ;
	    3: // Automat
	      "isAutPumping" := TRUE;
	      "isRecharging" := FALSE;
	      "isPumping" := False;
	      ;
	    4: // Ręczne
	      "isPumping" := TRUE;
	      "isRecharging" := FALSE;
	      "isAutPumping" := FALSE;
	      
	      ;
	    ELSE  // Statement section ELSE
	      "isRecharging" := FALSE;
	      "isPumping" := False;
	      "isAutPumping" := FALSE;
	      ;
	  END_CASE;
	  
	  
	END_REGION
	
	
	REGION Detekcja wybranego trybu sterowania zbiornikami 
	  // 
	  CASE "DB10_instance_SCADA".TrybSterowania OF
	    0:  // Wyłączone
	      "isDaily" := FALSE;
	      "isWeekiy" := FALSE;
	      "isManual" := FALSE;
	      ;
	    1:  // Dobowy
	      "isDaily" := TRUE;
	      "isWeekiy" := FALSE;
	      "isManual" := FALSE;
	      ;
	    2:  // Selektywny
	      "isDaily" := FALSE;
	      "isWeekiy" := TRUE;
	      "isManual" := FALSE;
	      ;
	    3:  // Ręczny
	      "isDaily" := FALSE;
	      "isWeekiy" := FALSE;
	      "isManual" := TRUE;
	      ;
	      
	    ELSE  // Statement section ELSE
	      "isDaily" := FALSE;
	      "isWeekiy" := FALSE;
	      "isManual" := FALSE;
	      ;
	  END_CASE;
	  
	  
	END_REGION
	
	
END_FUNCTION

FUNCTION_BLOCK "Nastawy_Parametrów_Sterownia"
TITLE = PARAMETRYZACJA ZBIORNIKÓW
{ S7_Optimized_Access := 'TRUE' }
AUTHOR : rtecmer
VERSION : 0.1
//Ustawienia trybu pracy zbiorników, parametrów podatawowych

BEGIN
	(*
	//=============================================================================
	//(JZWiK S.A Radosław Tecmer)
	//(c)Copyright (2022) All Rights Reserved
	//-----------------------------------------------------------------------------
	//Testowane z:   (system docelowy z  FW 4.4)
	//Pakiet inżynierski:   TIA Portal (V16 Update 6)
	//Ograniczenia:  ( - )
	//Wymagania:  (minimalne S7-1200 CPU 1215C FW 4.2 .)
	//Funkcjonalnośc: (Ustawienia parametrów sterowania zbiornikami.
	                   Aktywacja zbiornika (dołączenie do systemu w cykl automatyczny)
	//-----------------------------------------------------------------------------
	//Zmainy wprowadzone:
	//Wersja  Data       Osoba wprowadzająca zmiany - ekspert
	//01.00.00 08.09.2022 (Tecmer Radosław - twórca) Pieresza wersja 01.00.00
	//=============================================================================
	*)
	
	
	
	// zbiornuki wybór aktywnego
	REGION Zbiornik 1
	  // 
	  IF ("Hbit_Auto_Manu_Z1" = TRUE AND "Hbit_Auto_Manu_Z2" = TRUE)   THEN
	    // wtedy aktywney zbiornik 
	    "Parametryzacja"."Controls Tanks".aktywny_Zbiornik_1 := TRUE
	    ;
	  ELSE
	    "Parametryzacja"."Controls Tanks".aktywny_Zbiornik_1 := FALSE;
	  END_IF;
	  "Zmienne_sterujące_zbiorników".Zbiornik_1.active_Zb := "Parametryzacja"."Controls Tanks".aktywny_Zbiornik_1;
	  
	END_REGION
	
	
	REGION Zbiornik 2
	  // 
	  IF ("Hbit_Auto_Manu_Z3" = TRUE AND "Hbit_Auto_Manu_Z4" = TRUE) THEN
	    // wtedy aktywney zbiornik 
	    "Parametryzacja"."Controls Tanks".aktywny_Zbiornik_2 := TRUE
	    ;
	  ELSE
	    "Parametryzacja"."Controls Tanks".aktywny_Zbiornik_2 := FALSE;
	  END_IF;
	  "Zmienne_sterujące_zbiorników".Zbiornik_2.active_Zb := "Parametryzacja"."Controls Tanks".aktywny_Zbiornik_2;
	  
	END_REGION
	
	REGION Zbiornik 3
	  // 
	  IF ("Hbit_Auto_Manu_Z5" = TRUE AND "Hbit_Auto_Manu_Z6" = TRUE)  THEN
	    // wtedy aktywney zbiornik 
	    "Parametryzacja"."Controls Tanks".aktywny_Zbiornik_3 := TRUE
	    ;
	  ELSE
	    "Parametryzacja"."Controls Tanks".aktywny_Zbiornik_3 := FALSE;
	  END_IF;
	  "Zmienne_sterujące_zbiorników".Zbiornik_3.active_Zb := "Parametryzacja"."Controls Tanks".aktywny_Zbiornik_3;
	  
	END_REGION
	
	REGION Zbiornik 4
	  // 
	  IF ("Hbit_Auto_Manu_Z7" = TRUE AND "Hbit_Auto_Manu_Z8" = TRUE) THEN
	    // wtedy aktywney zbiornik 
	    "Parametryzacja"."Controls Tanks".aktywny_Zbiornik_4 := TRUE
	    ;
	  ELSE
	    "Parametryzacja"."Controls Tanks".aktywny_Zbiornik_4 := FALSE;
	  END_IF;
	  "Zmienne_sterujące_zbiorników".Zbiornik_4.active_Zb := "Parametryzacja"."Controls Tanks".aktywny_Zbiornik_4;
	  
	END_REGION
	
	
	
	REGION Aktywacja funkcji napełniania, 
	  // Gdy przynajmniej jeden zbiornik aktywny
	  IF "Parametryzacja"."Controls Tanks".aktywny_Zbiornik_1
	    OR "Parametryzacja"."Controls Tanks".aktywny_Zbiornik_2
	    OR "Parametryzacja"."Controls Tanks".aktywny_Zbiornik_3
	    OR "Parametryzacja"."Controls Tanks".aktywny_Zbiornik_4
	  THEN
	    // Wtedy aktywuj funcję 
	    "Parametryzacja"."Controls Tanks".aktywne_Napełnianie := TRUE;
	  
	  ELSE
	    "Parametryzacja"."Controls Tanks".aktywne_Napełnianie := FALSE;
	    ;
	  END_IF;
	  
	END_REGION
	
	REGION Aktywacja funkcji przetłaczania
	  // Gdy przynajmniej jeden zbiornik aktywny
	  IF ("Parametryzacja"."Controls Tanks".aktywny_Zbiornik_1
	    OR "Parametryzacja"."Controls Tanks".aktywny_Zbiornik_2
	    OR "Parametryzacja"."Controls Tanks".aktywny_Zbiornik_3
	    OR "Parametryzacja"."Controls Tanks".aktywny_Zbiornik_4)
	    AND "isPumping" 
	  THEN
	    // Wtedy aktywuj funcję 
	    "Parametryzacja"."Controls Tanks"."aktywne _Przetłaczanie" := TRUE;
	  ELSE
	    "Parametryzacja"."Controls Tanks"."aktywne _Przetłaczanie" := FALSE;
	    ;
	  END_IF;
	  
	END_REGION
	
	REGION Aktywacja funkcji dosilania
	  // Gdy przynajmniej jeden zbiornik aktywny
	  IF ("Parametryzacja"."Controls Tanks".aktywny_Zbiornik_1
	    OR "Parametryzacja"."Controls Tanks".aktywny_Zbiornik_2
	    OR "Parametryzacja"."Controls Tanks".aktywny_Zbiornik_3
	    OR "Parametryzacja"."Controls Tanks".aktywny_Zbiornik_4)
	    AND "isRecharging"
	  THEN
	    // Wtedy aktywuj funcję 
	    "Parametryzacja"."Controls Tanks".aktywne_Dosilanie := TRUE;
	  ELSE
	    "Parametryzacja"."Controls Tanks".aktywne_Dosilanie := FALSE;
	    ;
	  END_IF;
	  
	END_REGION
	
	
	
	
	
	
	
END_FUNCTION_BLOCK

FUNCTION "Konwerter zegarów" : Void   // FC19, LAD
TITLE = Konwersja DTL na Real
{ S7_Optimized_Access := 'TRUE' }
AUTHOR : rtecmer
VERSION : 0.1
// Funkcja konwersji czasu na wartość liczbowa
// stored: AutoNumber true, IsIECCheckEnabled false, SetENOAutomatically false, UDAEnableTagReadback false
   VAR_INPUT
      isPumping : Bool;   // sygnał ustawione przetłaczanie
      isRecharging : Bool;   // sygnał ustawione dosianie
      isAutpumping : Bool;   // sygnał usawione automatyczne sterowanie
   END_VAR
   VAR_TEMP
      timePumpingOn : Real;   // czas start przetłaczanie
      timePumpingOff : Real;   // czas stop przetłaczanie
      timeRechargingOn : Real;   // czas strat dosilanie
      timeRechargingoff : Real;   // czas stop dosilanie
   END_VAR
BEGIN

REGION Network 1: RTC local
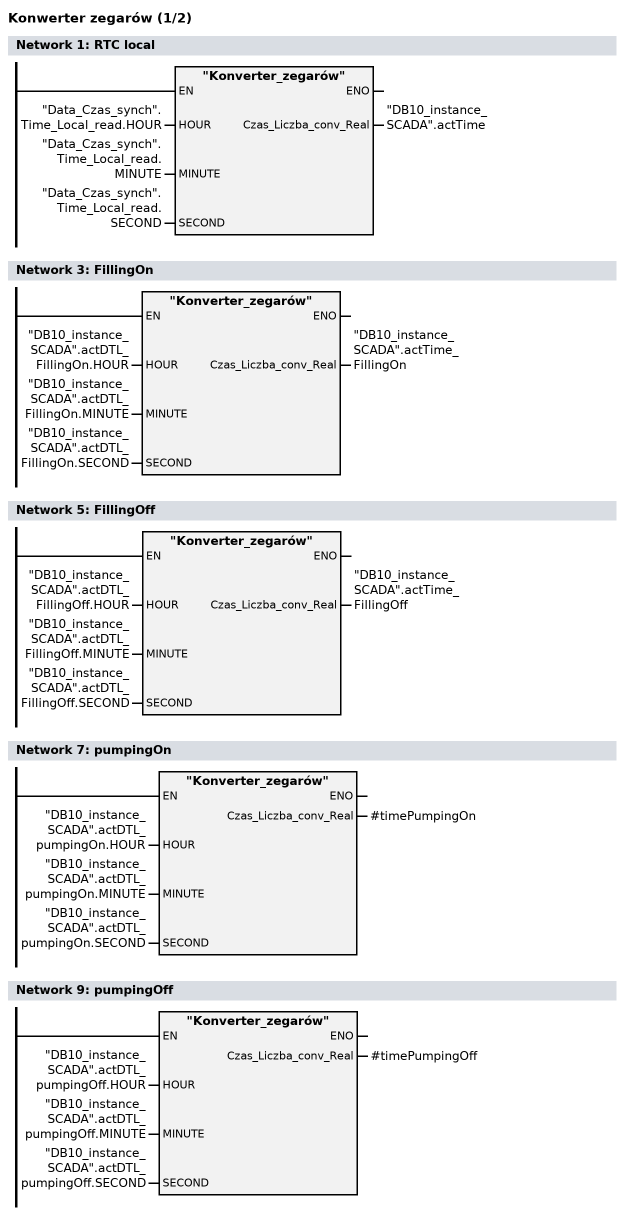
   RUNG wire#powerrail
      "Konverter_zegarów"(HOUR := "Data_Czas_synch".Time_Local_read.HOUR, MINUTE := "Data_Czas_synch".Time_Local_read.MINUTE, SECOND := "Data_Czas_synch".Time_Local_read.SECOND, Czas_Liczba_conv_Real => "DB10_instance_SCADA".actTime)
   END_RUNG
   // the same network as SCL:
   "Konverter_zegarów"(HOUR := "Data_Czas_synch".Time_Local_read.HOUR,
                       MINUTE := "Data_Czas_synch".Time_Local_read.MINUTE,
                       SECOND := "Data_Czas_synch".Time_Local_read.SECOND,
                       Czas_Liczba_conv_Real => "DB10_instance_SCADA".actTime);
END_REGION

REGION Network 3: FillingOn
   RUNG wire#powerrail
      "Konverter_zegarów"(HOUR := "DB10_instance_SCADA".actDTL_FillingOn.HOUR, MINUTE := "DB10_instance_SCADA".actDTL_FillingOn.MINUTE, SECOND := "DB10_instance_SCADA".actDTL_FillingOn.SECOND, Czas_Liczba_conv_Real => "DB10_instance_SCADA".actTime_FillingOn)
   END_RUNG
   // the same network as SCL:
   "Konverter_zegarów"(HOUR := "DB10_instance_SCADA".actDTL_FillingOn.HOUR,
                       MINUTE := "DB10_instance_SCADA".actDTL_FillingOn.MINUTE,
                       SECOND := "DB10_instance_SCADA".actDTL_FillingOn.SECOND,
                       Czas_Liczba_conv_Real => "DB10_instance_SCADA".actTime_FillingOn);
END_REGION

REGION Network 5: FillingOff
   RUNG wire#powerrail
      "Konverter_zegarów"(HOUR := "DB10_instance_SCADA".actDTL_FillingOff.HOUR, MINUTE := "DB10_instance_SCADA".actDTL_FillingOff.MINUTE, SECOND := "DB10_instance_SCADA".actDTL_FillingOff.SECOND, Czas_Liczba_conv_Real => "DB10_instance_SCADA".actTime_FillingOff)
   END_RUNG
   // the same network as SCL:
   "Konverter_zegarów"(HOUR := "DB10_instance_SCADA".actDTL_FillingOff.HOUR,
                       MINUTE := "DB10_instance_SCADA".actDTL_FillingOff.MINUTE,
                       SECOND := "DB10_instance_SCADA".actDTL_FillingOff.SECOND,
                       Czas_Liczba_conv_Real => "DB10_instance_SCADA".actTime_FillingOff);
END_REGION

REGION Network 7: pumpingOn
   RUNG wire#powerrail
      "Konverter_zegarów"(HOUR := "DB10_instance_SCADA".actDTL_pumpingOn.HOUR, MINUTE := "DB10_instance_SCADA".actDTL_pumpingOn.MINUTE, SECOND := "DB10_instance_SCADA".actDTL_pumpingOn.SECOND, Czas_Liczba_conv_Real => #timePumpingOn)
   END_RUNG
   // the same network as SCL:
   "Konverter_zegarów"(HOUR := "DB10_instance_SCADA".actDTL_pumpingOn.HOUR,
                       MINUTE := "DB10_instance_SCADA".actDTL_pumpingOn.MINUTE,
                       SECOND := "DB10_instance_SCADA".actDTL_pumpingOn.SECOND,
                       Czas_Liczba_conv_Real => #timePumpingOn);
END_REGION

REGION Network 9: pumpingOff
   RUNG wire#powerrail
      "Konverter_zegarów"(HOUR := "DB10_instance_SCADA".actDTL_pumpingOff.HOUR, MINUTE := "DB10_instance_SCADA".actDTL_pumpingOff.MINUTE, SECOND := "DB10_instance_SCADA".actDTL_pumpingOff.SECOND, Czas_Liczba_conv_Real => #timePumpingOff)
   END_RUNG
   // the same network as SCL:
   "Konverter_zegarów"(HOUR := "DB10_instance_SCADA".actDTL_pumpingOff.HOUR,
                       MINUTE := "DB10_instance_SCADA".actDTL_pumpingOff.MINUTE,
                       SECOND := "DB10_instance_SCADA".actDTL_pumpingOff.SECOND,
                       Czas_Liczba_conv_Real => #timePumpingOff);
END_REGION

REGION Network 11: RechargingOn
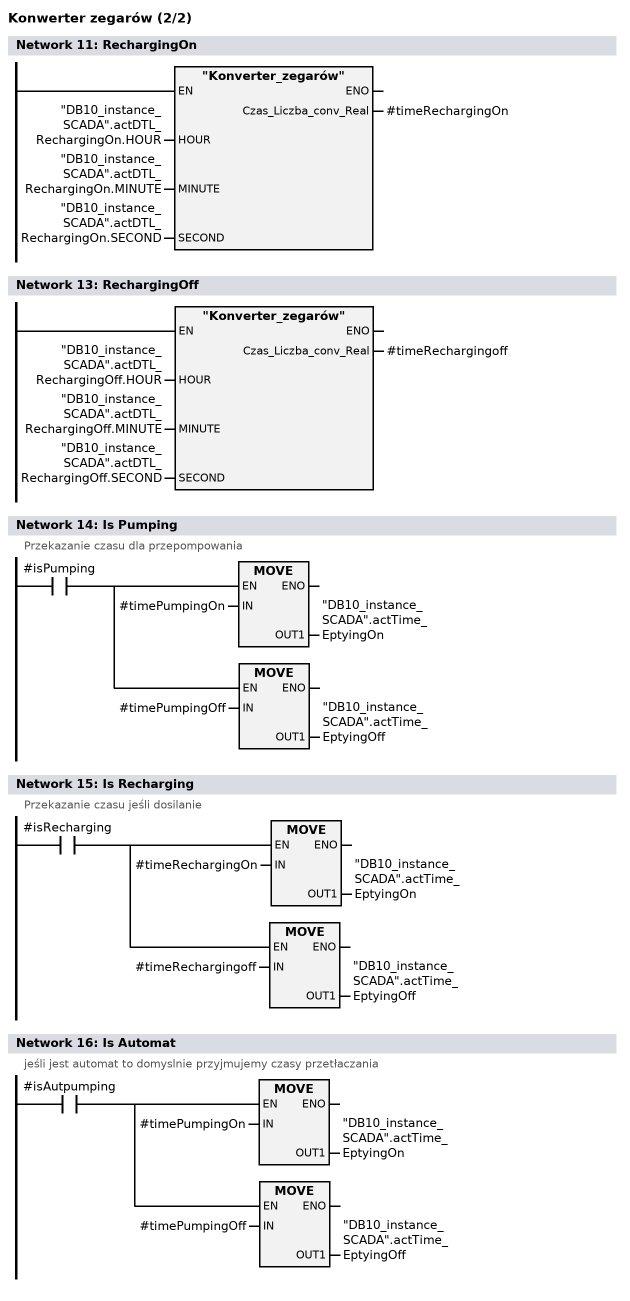
   RUNG wire#powerrail
      "Konverter_zegarów"(HOUR := "DB10_instance_SCADA".actDTL_RechargingOn.HOUR, MINUTE := "DB10_instance_SCADA".actDTL_RechargingOn.MINUTE, SECOND := "DB10_instance_SCADA".actDTL_RechargingOn.SECOND, Czas_Liczba_conv_Real => #timeRechargingOn)
   END_RUNG
   // the same network as SCL:
   "Konverter_zegarów"(HOUR := "DB10_instance_SCADA".actDTL_RechargingOn.HOUR,
                       MINUTE := "DB10_instance_SCADA".actDTL_RechargingOn.MINUTE,
                       SECOND := "DB10_instance_SCADA".actDTL_RechargingOn.SECOND,
                       Czas_Liczba_conv_Real => #timeRechargingOn);
END_REGION

REGION Network 13: RechargingOff
   RUNG wire#powerrail
      "Konverter_zegarów"(HOUR := "DB10_instance_SCADA".actDTL_RechargingOff.HOUR, MINUTE := "DB10_instance_SCADA".actDTL_RechargingOff.MINUTE, SECOND := "DB10_instance_SCADA".actDTL_RechargingOff.SECOND, Czas_Liczba_conv_Real => #timeRechargingoff)
   END_RUNG
   // the same network as SCL:
   "Konverter_zegarów"(HOUR := "DB10_instance_SCADA".actDTL_RechargingOff.HOUR,
                       MINUTE := "DB10_instance_SCADA".actDTL_RechargingOff.MINUTE,
                       SECOND := "DB10_instance_SCADA".actDTL_RechargingOff.SECOND,
                       Czas_Liczba_conv_Real => #timeRechargingoff);
END_REGION

REGION Network 14: Is Pumping
   // Przekazanie czasu dla przepompowania
   RUNG wire#powerrail
      Contact( #isPumping )
      wire#w1
      Move(in := #timePumpingOn, out1 => "DB10_instance_SCADA".actTime_EptyingOn)
   END_RUNG
   RUNG wire#w1
      Move(in := #timePumpingOff, out1 => "DB10_instance_SCADA".actTime_EptyingOff)
   END_RUNG
   // the same network as SCL:
   IF #isPumping THEN
       "DB10_instance_SCADA".actTime_EptyingOn := #timePumpingOn;
       "DB10_instance_SCADA".actTime_EptyingOff := #timePumpingOff;
   END_IF;
END_REGION

REGION Network 15: Is Recharging
   // Przekazanie czasu jeśli dosilanie
   RUNG wire#powerrail
      Contact( #isRecharging )
      wire#w1
      Move(in := #timeRechargingOn, out1 => "DB10_instance_SCADA".actTime_EptyingOn)
   END_RUNG
   RUNG wire#w1
      Move(in := #timeRechargingoff, out1 => "DB10_instance_SCADA".actTime_EptyingOff)
   END_RUNG
   // the same network as SCL:
   IF #isRecharging THEN
       "DB10_instance_SCADA".actTime_EptyingOn := #timeRechargingOn;
       "DB10_instance_SCADA".actTime_EptyingOff := #timeRechargingoff;
   END_IF;
END_REGION

REGION Network 16: Is Automat
   // jeśli jest automat to domyslnie przyjmujemy czasy przetłaczania
   RUNG wire#powerrail
      Contact( #isAutpumping )
      wire#w1
      Move(in := #timePumpingOn, out1 => "DB10_instance_SCADA".actTime_EptyingOn)
   END_RUNG
   RUNG wire#w1
      Move(in := #timePumpingOff, out1 => "DB10_instance_SCADA".actTime_EptyingOff)
   END_RUNG
   // the same network as SCL:
   IF #isAutpumping THEN
       "DB10_instance_SCADA".actTime_EptyingOn := #timePumpingOn;
       "DB10_instance_SCADA".actTime_EptyingOff := #timePumpingOff;
   END_IF;
END_REGION
END_FUNCTION

FUNCTION "Konverter_zegarów" : Void   // FC13, LAD
{ S7_Optimized_Access := 'FALSE' }
VERSION : 0.1
// stored: AutoNumber true, IsIECCheckEnabled false, SetENOAutomatically false, UDAEnableTagReadback false
   VAR_INPUT
      HOUR : USInt;   // Zmienna godzina z DTL
      MINUTE : USInt;   // Zmienna minuty z DTL
      SECOND : USInt;   // Zmienne sekundy z DTL
   END_VAR
   VAR_OUTPUT
      Czas_Liczba_conv_Real : Real;   // Liczba przedstawiająca czas 00:00:00 liczbowo 00.0000
   END_VAR
   VAR_TEMP
      zegar_H_pomocnicza : Real;   // pomocnicza do przekształcenia czasu z DLT do Real
      zegar_M_pomocnicza : Real;   // pomocnicza do przekształcenia czasu z DLT do Real
      zegar_S_pomocnicza : Real;   // pomocnicza do przekształcenia czasu z DLT do Real
      zegar_H_Uint : UInt;   // pomocnicza do przekształcenia czasu z DLT do Uint
      zegar_M_Uint : UInt;   // pomocnicza do przekształcenia czasu z DLT do Uint
      zegar_S_Uint : UInt;   // pomocnicza do przekształcenia czasu z DLT do Uint
   END_VAR
BEGIN

REGION Network 1: Wyodrębnienie zegara z danej DTL czasu lokalnego
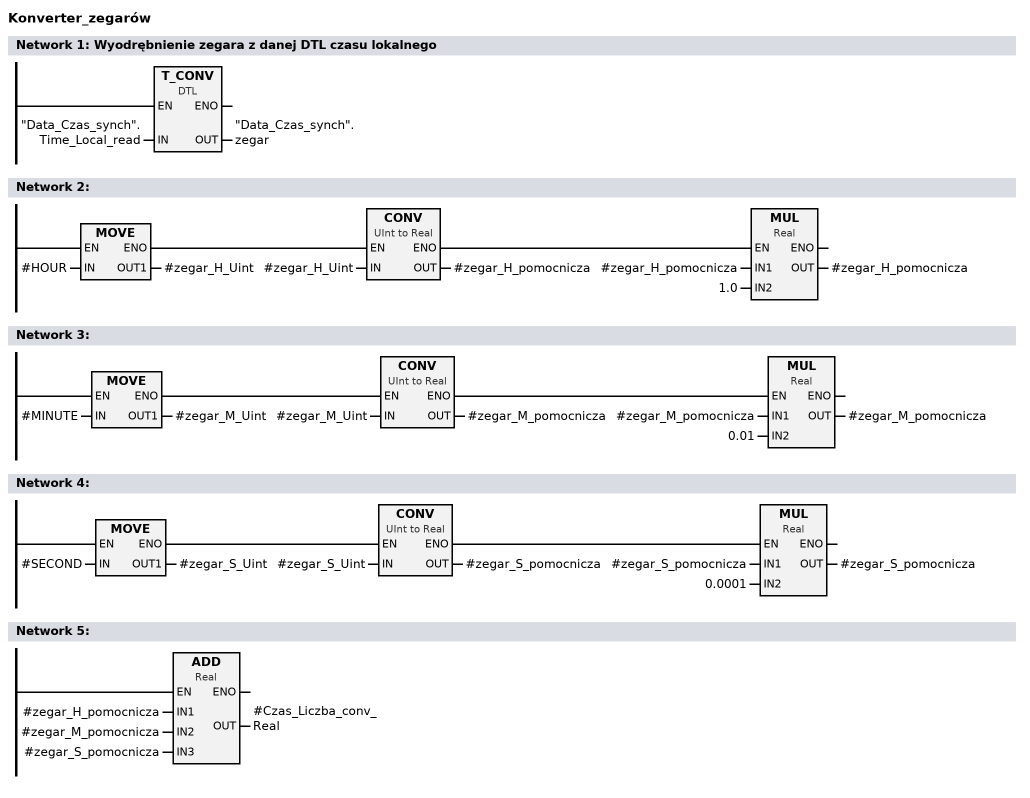
   RUNG wire#powerrail
      { S7_Templates := "[src_type := DTL, dest_type := Time_Of_Day]" } T_CONV(IN := "Data_Czas_synch".Time_Local_read, OUT => "Data_Czas_synch".zegar)
   END_RUNG
   // the same network as SCL:
   T_CONV(IN := "Data_Czas_synch".Time_Local_read, OUT => "Data_Czas_synch".zegar);
END_REGION

REGION Network 2
   RUNG wire#powerrail
      { S7_GenerateENO := "TRUE" } Move(in := #HOUR, out1 => #zegar_H_Uint)
      { S7_Templates := "[SrcType := UInt, DestType := Real]"; S7_GenerateENO := "TRUE" } Convert(in := #zegar_H_Uint, out => #zegar_H_pomocnicza)
      { S7_Templates := "SrcType := Real"; S7_GenerateENO := "TRUE" } Mul(in1 := #zegar_H_pomocnicza, in2 := 1.0, out => #zegar_H_pomocnicza)
   END_RUNG
   // the same network as SCL:
   // ENO of a box is taken as its EN; it also drops when the box reports an error
   #zegar_H_Uint := #HOUR;
   #zegar_H_pomocnicza := UINT_TO_REAL(#zegar_H_Uint);
   #zegar_H_pomocnicza := #zegar_H_pomocnicza * 1.0;
END_REGION

REGION Network 3
   RUNG wire#powerrail
      { S7_GenerateENO := "TRUE" } Move(in := #MINUTE, out1 => #zegar_M_Uint)
      { S7_Templates := "[SrcType := UInt, DestType := Real]"; S7_GenerateENO := "TRUE" } Convert(in := #zegar_M_Uint, out => #zegar_M_pomocnicza)
      { S7_Templates := "SrcType := Real"; S7_GenerateENO := "TRUE" } Mul(in1 := #zegar_M_pomocnicza, in2 := 0.01, out => #zegar_M_pomocnicza)
   END_RUNG
   // the same network as SCL:
   // ENO of a box is taken as its EN; it also drops when the box reports an error
   #zegar_M_Uint := #MINUTE;
   #zegar_M_pomocnicza := UINT_TO_REAL(#zegar_M_Uint);
   #zegar_M_pomocnicza := #zegar_M_pomocnicza * 0.01;
END_REGION

REGION Network 4
   RUNG wire#powerrail
      { S7_GenerateENO := "TRUE" } Move(in := #SECOND, out1 => #zegar_S_Uint)
      { S7_Templates := "[SrcType := UInt, DestType := Real]"; S7_GenerateENO := "TRUE" } Convert(in := #zegar_S_Uint, out => #zegar_S_pomocnicza)
      { S7_Templates := "SrcType := Real"; S7_GenerateENO := "TRUE" } Mul(in1 := #zegar_S_pomocnicza, in2 := 0.0001, out => #zegar_S_pomocnicza)
   END_RUNG
   // the same network as SCL:
   // ENO of a box is taken as its EN; it also drops when the box reports an error
   #zegar_S_Uint := #SECOND;
   #zegar_S_pomocnicza := UINT_TO_REAL(#zegar_S_Uint);
   #zegar_S_pomocnicza := #zegar_S_pomocnicza * 0.0001;
END_REGION

REGION Network 5
   RUNG wire#powerrail
      { S7_Templates := "SrcType := Real"; S7_GenerateENO := "TRUE" } Add(in1 := #zegar_H_pomocnicza, in2 := #zegar_M_pomocnicza, in3 := #zegar_S_pomocnicza, out => #Czas_Liczba_conv_Real)
   END_RUNG
   // the same network as SCL:
   #Czas_Liczba_conv_Real := #zegar_H_pomocnicza + #zegar_M_pomocnicza + #zegar_S_pomocnicza;
END_REGION
END_FUNCTION

FUNCTION "Czyszczenie_błednych_wpisów" : Void
TITLE = Korekta błednego wpisu
{ S7_Optimized_Access := 'TRUE' }
AUTHOR : rtecmer
VERSION : 0.1
//Program kontroluje błedny wpis wartości poza granicą liczby określającej czas (godziny, minuty) W razie wpisania złej wartości wypełna komurkę zerami

BEGIN
	(*
	//=============================================================================
	//(JZWiK S.A Radosław Tecmer)
	//(c)Copyright (2022) All Rights Reserved
	//-----------------------------------------------------------------------------
	//Testowane z:   (system docelowy z  FW 4.4)
	//Pakiet inżynierski:   TIA Portal (V16 Update 5)
	//Ograniczenia:  ( - )
	//Wymagania:  (minimalne S7-1200 CPU 1215C FW 4.2 .)
	//Funkcjonalnośc: (Kontrola błednego wpisy wartości liczbowej czasu, wartości.
	                   Jeśli wartość poza zakresem wypełnieni komórki zerami)
	//-----------------------------------------------------------------------------
	//Zmainy wprowadzone:
	//Wersja  Data       Osoba wprowadzająca zmiany - ekspert
	//01.00.00 05.05.2022 (Tecmer Radosław - twórca) Pieresza wersja 01.00.00
	//=============================================================================
	*)
	
	
	
	//poziomu
	
	//napełnianie
	IF "DB10_instance_SCADA".setPoziomNapełniania < 0
	  OR "DB10_instance_SCADA".setPoziomNapełniania > 1000
	  OR "dbHold_Sending".data.stat.control.set_poziom_napełniania <0
	  OR "dbHold_Sending".data.stat.control.set_poziom_napełniania > 1000
	THEN
	  // wypełnij zerami
	  "DB10_instance_SCADA".setPoziomNapełniania := 0;
	  "tempdbHold_SendingTCP".sterowanie.set_poziom_napełniania := 0;
	  "dbHold_Sending".data.stat.control.set_poziom_napełniania := 0;
	  "dbHold_download".sterowanie.set_poziom_napełniania := 0;
	  ;
	END_IF;
	
	//opróżnianie
	IF "DB10_instance_SCADA".setPoziomOpróżnianai < 0
	  OR "DB10_instance_SCADA".setPoziomOpróżnianai > 1000
	  OR "dbHold_Sending".data.stat.control.set_poziom_opróżniania < 0
	  OR "dbHold_Sending".data.stat.control.set_poziom_opróżniania > 1000
	  OR "DB10_instance_SCADA".setPoziomOpróżnianai >= "DB10_instance_SCADA".setPoziomNapełniania
	  OR "dbHold_Sending".data.stat.control.set_poziom_opróżniania >= "dbHold_Sending".data.stat.control.set_poziom_napełniania
	THEN
	  // wypełnij zerami
	  "DB10_instance_SCADA".setPoziomOpróżnianai := 0;
	  "tempdbHold_SendingTCP".sterowanie.set_poziom_opróżniania := 0;
	  "dbHold_Sending".data.stat.control.set_poziom_opróżniania := 0;
	  ;
	END_IF;
	
	
	// Zadawane położenie zasuwy Z10 
	IF "DB10_instance_SCADA".setPołożenieZ10 < 0
	  OR "DB10_instance_SCADA".setPołożenieZ10 > 100
	  OR "dbHold_Sending".data.stat.control.control_2.set_położenie_Z10 < 0
	  OR "dbHold_Sending".data.stat.control.control_2.set_położenie_Z10 > 100
	THEN
	  // wypełnij zerami      
	  "DB10_instance_SCADA".setPołożenieZ10 := 0;
	  "tempdbHold_SendingTCP".sterowanie.set_położenie_Z10 := 0;
	  "dbHold_Sending".data.stat.control.control_2.set_położenie_Z10 := 0;
	  ;
	END_IF;
	
	// Strategia sterowania zbiornikami
	
	
	// Czasy 
	// napełnianie
	
	IF "DB10_instance_SCADA".actDTL_FillingOn.HOUR < 0
	  OR "DB10_instance_SCADA".actDTL_FillingOn.HOUR > 23
	  OR "tempdbHold_SendingTCP".start_napełnianie.HOUR < 0
	  OR "tempdbHold_SendingTCP".start_napełnianie.HOUR > 23
	THEN
	  // wypełnij zerami
	  "DB10_instance_SCADA".actDTL_FillingOn.HOUR := 0;
	  "tempdbHold_SendingTCP".start_napełnianie.HOUR := 0;
	  "dbHold_download".SendingTimes.start_napełnianie.HOUR := 0;
	  "dbHold_Sending".data."Time".start_napełnianie.HOUR:= 0;
	  ;
	END_IF;
	
	IF "DB10_instance_SCADA".actDTL_FillingOn.MINUTE < 0
	  OR "DB10_instance_SCADA".actDTL_FillingOn.MINUTE > 60
	  OR "dbHold_Sending".data."Time".start_napełnianie.MINUTE < 0
	  OR "dbHold_Sending".data."Time".start_napełnianie.MINUTE > 60
	THEN
	  // wypełnij zerami
	  "DB10_instance_SCADA".actDTL_FillingOn.MINUTE := 0;
	  "tempdbHold_SendingTCP".start_napełnianie.MINUTE := 0;
	  "dbHold_Sending".data."Time".start_napełnianie.MINUTE := 0;
	  ;
	END_IF;
	
	// opróżnianie
	IF "DB10_instance_SCADA".actDTL_FillingOff.HOUR < 0
	  OR "DB10_instance_SCADA".actDTL_FillingOff.HOUR > 23
	  OR "dbHold_Sending".data."Time".Stop_napełnianie.HOUR < 0
	  OR "dbHold_Sending".data."Time".Stop_napełnianie.HOUR > 23
	THEN
	  // wypełnij zerami
	  "DB10_instance_SCADA".actDTL_FillingOff.HOUR := 0;
	  "tempdbHold_SendingTCP".Stop_napełnianie.HOUR := 0;
	  "dbHold_Sending".data."Time".Stop_napełnianie.HOUR := 0;
	  ;
	END_IF;
	
	IF "DB10_instance_SCADA".actDTL_FillingOff.MINUTE < 0
	  OR "DB10_instance_SCADA".actDTL_FillingOff.MINUTE > 60
	  OR "dbHold_Sending".data."Time".Stop_napełnianie.MINUTE < 0
	  OR "dbHold_Sending".data."Time".Stop_napełnianie.MINUTE > 60
	THEN
	  // wypełnij zerami
	  "DB10_instance_SCADA".actDTL_FillingOff.MINUTE := 0;
	  "tempdbHold_SendingTCP".Stop_napełnianie.MINUTE := 0;
	  "dbHold_Sending".data."Time".Stop_napełnianie.MINUTE := 0;
	  ;
	END_IF;
	
	// przetłaczanie
	IF "DB10_instance_SCADA".actDTL_pumpingOn.HOUR < 0
	  OR "DB10_instance_SCADA".actDTL_pumpingOn.HOUR > 23
	  OR "dbHold_Sending".data."Time".Start_przetłaczanie_1.HOUR < 0
	  OR "dbHold_Sending".data."Time".Start_przetłaczanie_1.HOUR > 23
	THEN
	  // wypełnij zerami
	  "DB10_instance_SCADA".actDTL_pumpingOn.HOUR := 0;
	  "tempdbHold_SendingTCP".Start_przetłaczanie_1.HOUR := 0;
	  "dbHold_Sending".data."Time".Start_przetłaczanie_1.HOUR := 0;
	  ;
	END_IF;
	
	IF "DB10_instance_SCADA".actDTL_pumpingOn.MINUTE < 0
	  OR "DB10_instance_SCADA".actDTL_pumpingOn.MINUTE > 60
	  OR "dbHold_Sending".data."Time".Start_przetłaczanie_1.MINUTE < 0
	  OR "dbHold_Sending".data."Time".Start_przetłaczanie_1.MINUTE > 60
	THEN
	  // wypełnij zerami
	  "DB10_instance_SCADA".actDTL_pumpingOn.MINUTE := 0;
	  "tempdbHold_SendingTCP".Start_przetłaczanie_1.MINUTE := 0;
	  "dbHold_Sending".data."Time".Start_przetłaczanie_1.MINUTE := 0;
	  ;
	END_IF;
	
	// stop przetłaczanie
	IF "DB10_instance_SCADA".actDTL_pumpingOff.HOUR < 0
	  OR "DB10_instance_SCADA".actDTL_pumpingOff.HOUR > 23
	  OR "dbHold_Sending".data."Time".Stop_przetłaczanie_1.HOUR < 0
	  OR "dbHold_Sending".data."Time".Stop_przetłaczanie_1.HOUR > 23
	THEN
	  // wypełnij zerami
	  "DB10_instance_SCADA".actDTL_pumpingOff.HOUR := 0;
	  "tempdbHold_SendingTCP".Stop_przetłaczanie_1.HOUR := 0;
	  "dbHold_Sending".data."Time".Stop_przetłaczanie_1.HOUR := 0;
	  ;
	END_IF;
	
	IF "DB10_instance_SCADA".actDTL_pumpingOff.MINUTE < 0
	  OR "DB10_instance_SCADA".actDTL_pumpingOff.MINUTE > 60
	  OR "dbHold_Sending".data."Time".Stop_przetłaczanie_1.MINUTE < 0
	  OR "dbHold_Sending".data."Time".Stop_przetłaczanie_1.MINUTE > 60
	THEN
	  // wypełnij zerami
	  "DB10_instance_SCADA".actDTL_pumpingOff.MINUTE := 0;
	  "tempdbHold_SendingTCP".Stop_przetłaczanie_1.MINUTE := 0;
	  "dbHold_Sending".data."Time".Stop_przetłaczanie_1.MINUTE := 0;
	  ;
	END_IF;
	
